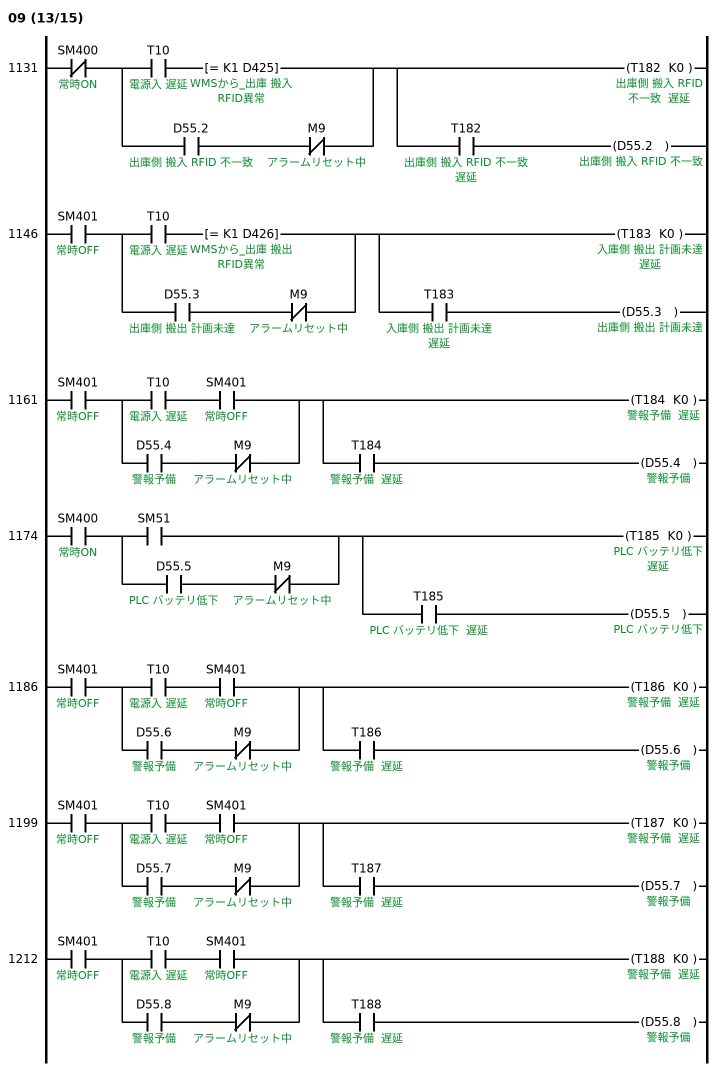
1131  LDI     SM400  ; 常時ON
      LD      T10  ; 電源入 遅延
      AND=    K1 D425  ; WMSから_出庫 搬入 RFID異常
      LD      D55.2  ; 出庫側 搬入 RFID 不一致
      ANI     M9  ; アラームリセット中
      ORB
      ANB
      OUT     T182 K0  ; 出庫側 搬入 RFID 不一致  遅延
      AND     T182  ; 出庫側 搬入 RFID 不一致  遅延
      OUT     D55.2  ; 出庫側 搬入 RFID 不一致
1146  LD      SM401  ; 常時OFF
      LD      T10  ; 電源入 遅延
      AND=    K1 D426  ; WMSから_出庫 搬出 RFID異常
      LD      D55.3  ; 出庫側 搬出 計画未達
      ANI     M9  ; アラームリセット中
      ORB
      ANB
      OUT     T183 K0  ; 入庫側 搬出 計画未達  遅延
      AND     T183  ; 入庫側 搬出 計画未達  遅延
      OUT     D55.3  ; 出庫側 搬出 計画未達
1161  LD      SM401  ; 常時OFF
      LD      T10  ; 電源入 遅延
      AND     SM401  ; 常時OFF
      LD      D55.4  ; 警報予備
      ANI     M9  ; アラームリセット中
      ORB
      ANB
      OUT     T184 K0  ; 警報予備  遅延
      AND     T184  ; 警報予備  遅延
      OUT     D55.4  ; 警報予備
1174  LD      SM400  ; 常時ON
      LD      SM51
      LD      D55.5  ; PLC バッテリ低下
      ANI     M9  ; アラームリセット中
      ORB
      ANB
      OUT     T185 K0  ; PLC バッテリ低下  遅延
      AND     T185  ; PLC バッテリ低下  遅延
      OUT     D55.5  ; PLC バッテリ低下
1186  LD      SM401  ; 常時OFF
      LD      T10  ; 電源入 遅延
      AND     SM401  ; 常時OFF
      LD      D55.6  ; 警報予備
      ANI     M9  ; アラームリセット中
      ORB
      ANB
      OUT     T186 K0  ; 警報予備  遅延
      AND     T186  ; 警報予備  遅延
      OUT     D55.6  ; 警報予備
1199  LD      SM401  ; 常時OFF
      LD      T10  ; 電源入 遅延
      AND     SM401  ; 常時OFF
      LD      D55.7  ; 警報予備
      ANI     M9  ; アラームリセット中
      ORB
      ANB
      OUT     T187 K0  ; 警報予備  遅延
      AND     T187  ; 警報予備  遅延
      OUT     D55.7  ; 警報予備
1212  LD      SM401  ; 常時OFF
      LD      T10  ; 電源入 遅延
      AND     SM401  ; 常時OFF
      LD      D55.8  ; 警報予備
      ANI     M9  ; アラームリセット中
      ORB
      ANB
      OUT     T188 K0  ; 警報予備  遅延
      AND     T188  ; 警報予備  遅延
      OUT     D55.8  ; 警報予備
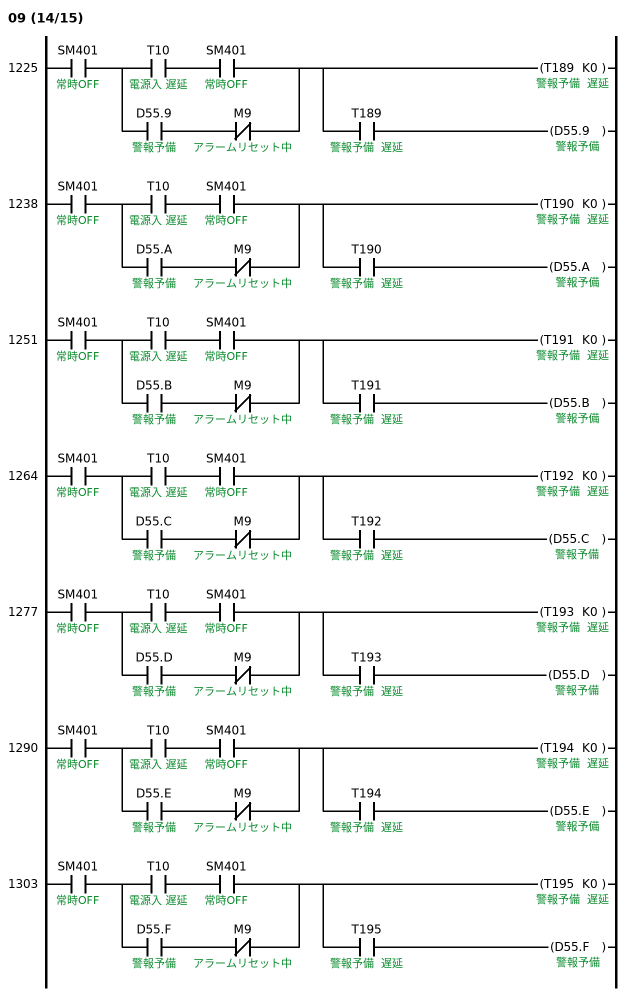
1225  LD      SM401  ; 常時OFF
      LD      T10  ; 電源入 遅延
      AND     SM401  ; 常時OFF
      LD      D55.9  ; 警報予備
      ANI     M9  ; アラームリセット中
      ORB
      ANB
      OUT     T189 K0  ; 警報予備  遅延
      AND     T189  ; 警報予備  遅延
      OUT     D55.9  ; 警報予備
1238  LD      SM401  ; 常時OFF
      LD      T10  ; 電源入 遅延
      AND     SM401  ; 常時OFF
      LD      D55.A  ; 警報予備
      ANI     M9  ; アラームリセット中
      ORB
      ANB
      OUT     T190 K0  ; 警報予備  遅延
      AND     T190  ; 警報予備  遅延
      OUT     D55.A  ; 警報予備
1251  LD      SM401  ; 常時OFF
      LD      T10  ; 電源入 遅延
      AND     SM401  ; 常時OFF
      LD      D55.B  ; 警報予備
      ANI     M9  ; アラームリセット中
      ORB
      ANB
      OUT     T191 K0  ; 警報予備  遅延
      AND     T191  ; 警報予備  遅延
      OUT     D55.B  ; 警報予備
1264  LD      SM401  ; 常時OFF
      LD      T10  ; 電源入 遅延
      AND     SM401  ; 常時OFF
      LD      D55.C  ; 警報予備
      ANI     M9  ; アラームリセット中
      ORB
      ANB
      OUT     T192 K0  ; 警報予備  遅延
      AND     T192  ; 警報予備  遅延
      OUT     D55.C  ; 警報予備
1277  LD      SM401  ; 常時OFF
      LD      T10  ; 電源入 遅延
      AND     SM401  ; 常時OFF
      LD      D55.D  ; 警報予備
      ANI     M9  ; アラームリセット中
      ORB
      ANB
      OUT     T193 K0  ; 警報予備  遅延
      AND     T193  ; 警報予備  遅延
      OUT     D55.D  ; 警報予備
1290  LD      SM401  ; 常時OFF
      LD      T10  ; 電源入 遅延
      AND     SM401  ; 常時OFF
      LD      D55.E  ; 警報予備
      ANI     M9  ; アラームリセット中
      ORB
      ANB
      OUT     T194 K0  ; 警報予備  遅延
      AND     T194  ; 警報予備  遅延
      OUT     D55.E  ; 警報予備
1303  LD      SM401  ; 常時OFF
      LD      T10  ; 電源入 遅延
      AND     SM401  ; 常時OFF
      LD      D55.F  ; 警報予備
      ANI     M9  ; アラームリセット中
      ORB
      ANB
      OUT     T195 K0  ; 警報予備  遅延
      AND     T195  ; 警報予備  遅延
      OUT     D55.F  ; 警報予備
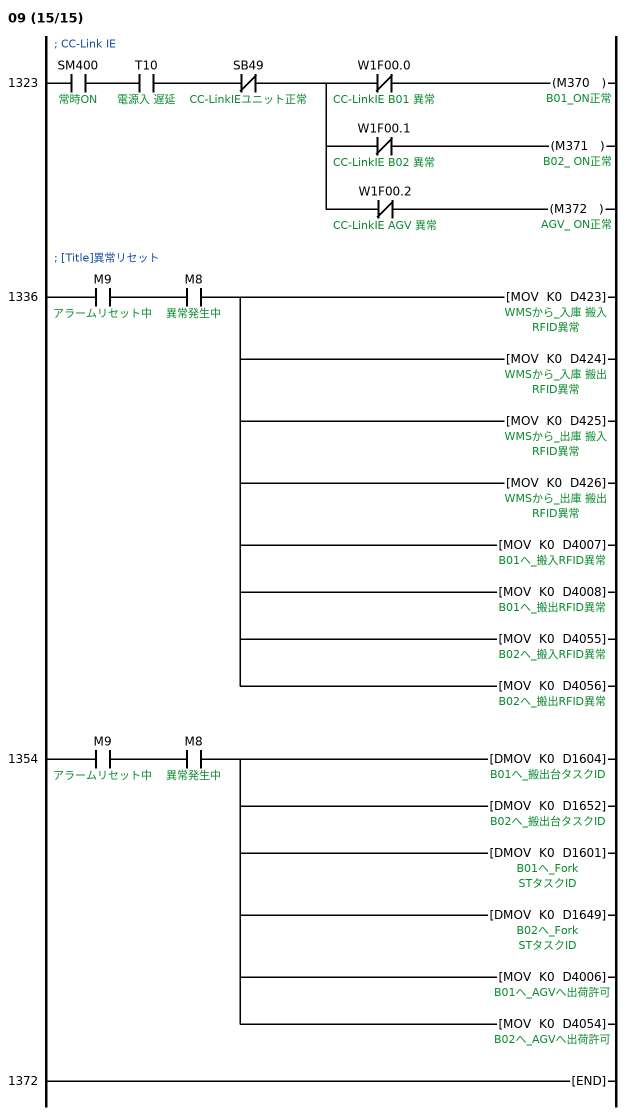
; CC-Link IE
1323  LD      SM400  ; 常時ON
      AND     T10  ; 電源入 遅延
      ANI     SB49  ; CC-LinkIEユニット正常
      MPS
      ANI     W1F00.0  ; CC-LinkIE B01 異常
      OUT     M370  ; B01_ON正常
      MRD
      ANI     W1F00.1  ; CC-LinkIE B02 異常
      OUT     M371  ; B02_ ON正常
      MPP
      ANI     W1F00.2  ; CC-LinkIE AGV 異常
      OUT     M372  ; AGV_ ON正常
; [Title]異常リセット
1336  LD      M9  ; アラームリセット中
      AND     M8  ; 異常発生中
      MOV     K0 D423
      MOV     K0 D424
      MOV     K0 D425
      MOV     K0 D426
      MOV     K0 D4007  ; B01へ_搬入RFID異常
      MOV     K0 D4008  ; B01へ_搬出RFID異常
      MOV     K0 D4055  ; B02へ_搬入RFID異常
      MOV     K0 D4056  ; B02へ_搬出RFID異常
1354  LD      M9  ; アラームリセット中
      AND     M8  ; 異常発生中
      DMOV    K0 D1604  ; B01へ_搬出台タスクID
      DMOV    K0 D1652  ; B02へ_搬出台タスクID
      DMOV    K0 D1601  ; B01へ_ForkSTタスクID
      DMOV    K0 D1649  ; B02へ_ForkSTタスクID
      MOV     K0 D4006  ; B01へ_AGVへ出荷許可
      MOV     K0 D4054  ; B02へ_AGVへ出荷許可
1372  END
END_PROGRAM

PROGRAM 10  // MAIN
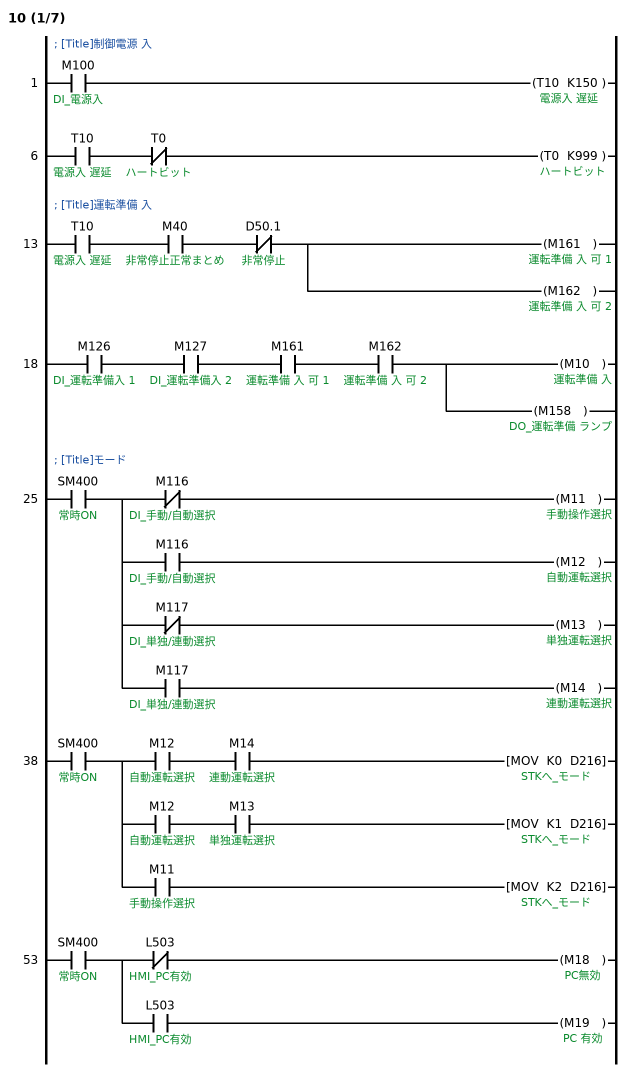
; [Title]制御電源 入
1     LD      M100  ; DI_電源入
      OUT     T10 K150  ; 電源入 遅延
6     LD      T10  ; 電源入 遅延
      ANI     T0  ; ハートビット
      OUT     T0 K999  ; ハートビット
; [Title]運転準備 入
13    LD      T10  ; 電源入 遅延
      AND     M40  ; 非常停止正常まとめ
      ANI     D50.1  ; 非常停止
      OUT     M161  ; 運転準備 入 可 1
      OUT     M162  ; 運転準備 入 可 2
18    LD      M126  ; DI_運転準備入 1
      AND     M127  ; DI_運転準備入 2
      AND     M161  ; 運転準備 入 可 1
      AND     M162  ; 運転準備 入 可 2
      OUT     M10  ; 運転準備 入
      OUT     M158  ; DO_運転準備 ランプ
; [Title]モード
25    LD      SM400  ; 常時ON
      MPS
      ANI     M116  ; DI_手動/自動選択
      OUT     M11  ; 手動操作選択
      MRD
      AND     M116  ; DI_手動/自動選択
      OUT     M12  ; 自動運転選択
      MRD
      ANI     M117  ; DI_単独/連動選択
      OUT     M13  ; 単独運転選択
      MPP
      AND     M117  ; DI_単独/連動選択
      OUT     M14  ; 連動運転選択
38    LD      SM400  ; 常時ON
      MPS
      AND     M12  ; 自動運転選択
      AND     M14  ; 連動運転選択
      MOV     K0 D216  ; STKへ_モード
      MRD
      AND     M12  ; 自動運転選択
      AND     M13  ; 単独運転選択
      MOV     K1 D216
      MPP
      AND     M11  ; 手動操作選択
      MOV     K2 D216
53    LD      SM400  ; 常時ON
      MPS
      ANI     L503  ; HMI_PC有効
      OUT     M18  ; PC無効
      MPP
      AND     L503  ; HMI_PC有効
      OUT     M19  ; PC 有効
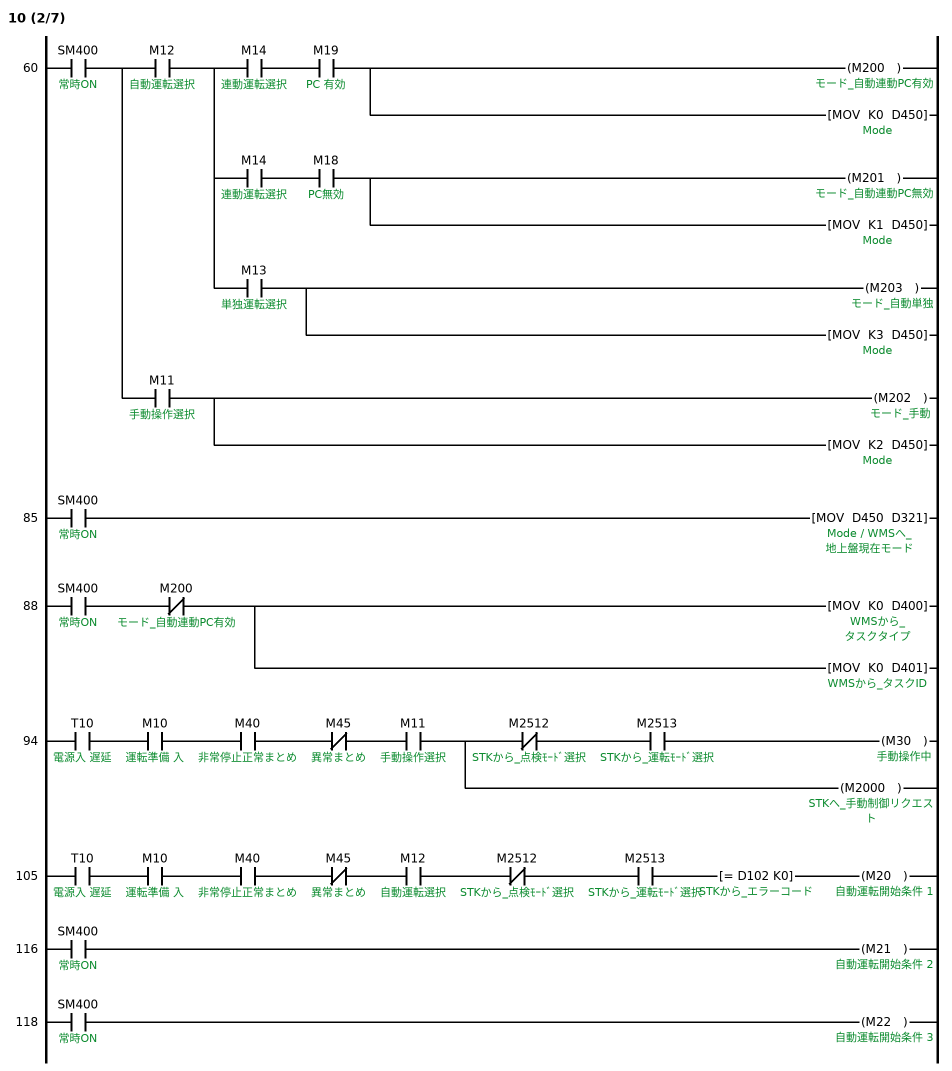
60    LD      SM400  ; 常時ON
      MPS
      AND     M12  ; 自動運転選択
      MPS
      AND     M14  ; 連動運転選択
      AND     M19  ; PC 有効
      OUT     M200  ; モード_自動連動PC有効
      MOV     K0 D450  ; Mode
      MRD
      AND     M14  ; 連動運転選択
      AND     M18  ; PC無効
      OUT     M201  ; モード_自動連動PC無効
      MOV     K1 D450
      MPP
      AND     M13  ; 単独運転選択
      OUT     M203  ; モード_自動単独
      MOV     K3 D450
      MPP
      AND     M11  ; 手動操作選択
      OUT     M202  ; モード_手動
      MOV     K2 D450
85    LD      SM400  ; 常時ON
      MOV     D450 D321  ; WMSへ_地上盤現在モード
88    LD      SM400  ; 常時ON
      ANI     M200  ; モード_自動連動PC有効
      MOV     K0 D400  ; WMSから_タスクタイプ
      MOV     K0 D401  ; WMSから_タスクID
94    LD      T10  ; 電源入 遅延
      AND     M10  ; 運転準備 入
      AND     M40  ; 非常停止正常まとめ
      ANI     M45  ; 異常まとめ
      AND     M11  ; 手動操作選択
      MPS
      ANI     M2512  ; STKから_点検ﾓｰﾄﾞ選択
      AND     M2513  ; STKから_運転ﾓｰﾄﾞ選択
      OUT     M30  ; 手動操作中
      MPP
      OUT     M2000  ; STKへ_手動制御リクエスト
105   LD      T10  ; 電源入 遅延
      AND     M10  ; 運転準備 入
      AND     M40  ; 非常停止正常まとめ
      ANI     M45  ; 異常まとめ
      AND     M12  ; 自動運転選択
      ANI     M2512  ; STKから_点検ﾓｰﾄﾞ選択
      AND     M2513  ; STKから_運転ﾓｰﾄﾞ選択
      AND=    D102 K0  ; STKから_エラーコード
      OUT     M20  ; 自動運転開始条件 1
116   LD      SM400  ; 常時ON
      OUT     M21  ; 自動運転開始条件 2
118   LD      SM400  ; 常時ON
      OUT     M22  ; 自動運転開始条件 3
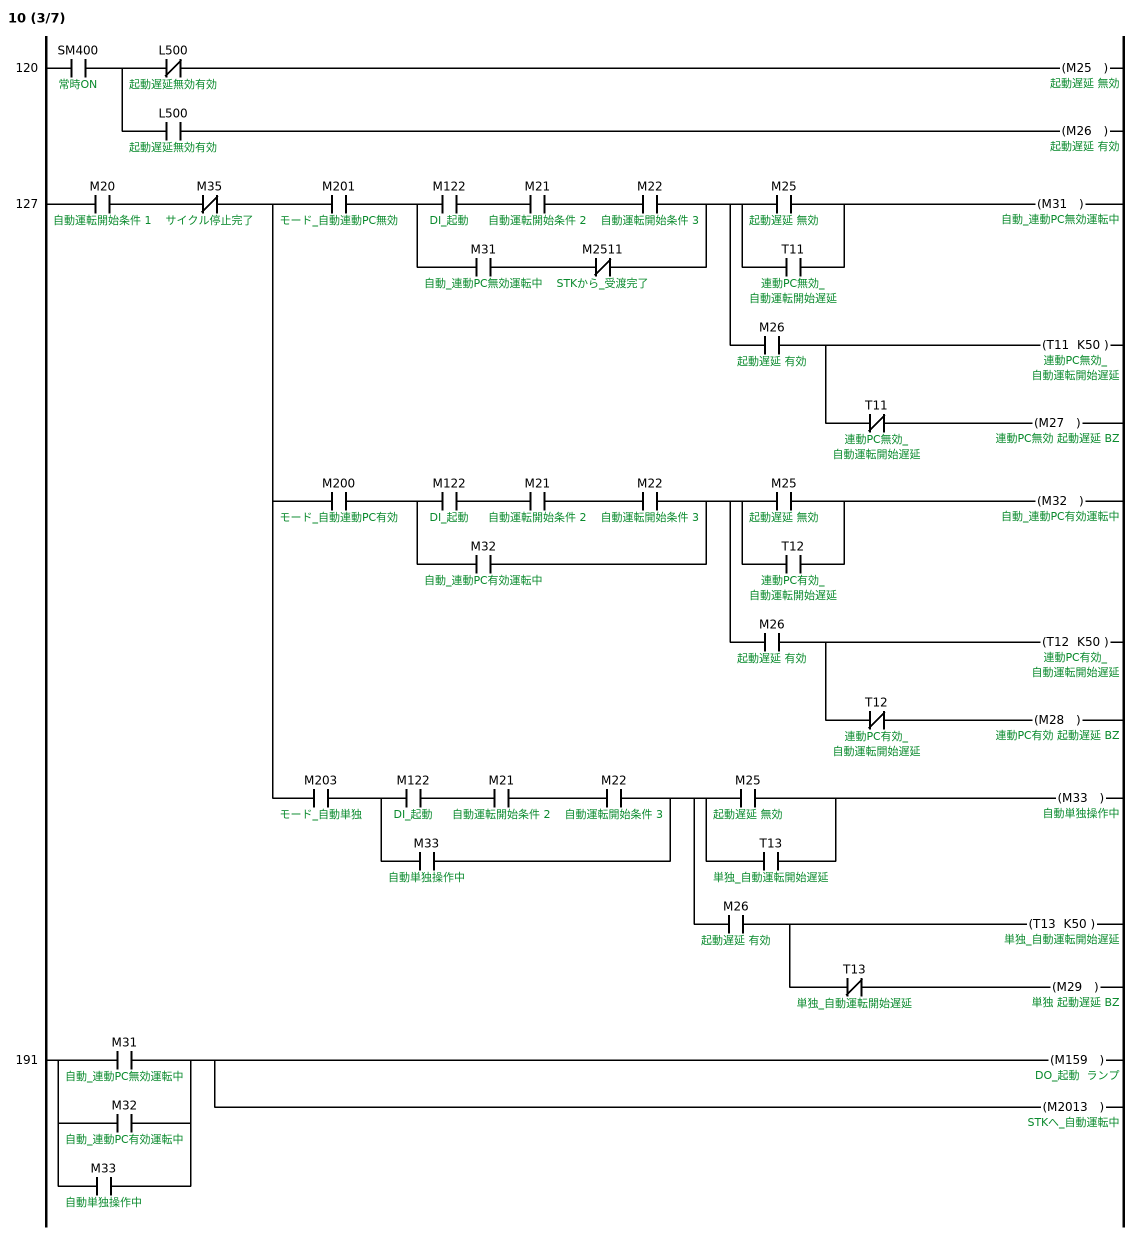
120   LD      SM400  ; 常時ON
      MPS
      ANI     L500  ; 起動遅延無効有効
      OUT     M25  ; 起動遅延 無効
      MPP
      AND     L500  ; 起動遅延無効有効
      OUT     M26  ; 起動遅延 有効
127   LD      M20  ; 自動運転開始条件 1
      ANI     M35  ; サイクル停止完了
      MPS
      AND     M201  ; モード_自動連動PC無効
      LD      M122  ; DI_起動
      AND     M21  ; 自動運転開始条件 2
      AND     M22  ; 自動運転開始条件 3
      LD      M31  ; 自動_連動PC無効運転中
      ANI     M2511  ; STKから_受渡完了
      ORB
      ANB
      MPS
      LD      M25  ; 起動遅延 無効
      OR      T11  ; 連動PC無効_自動運転開始遅延
      ANB
      OUT     M31  ; 自動_連動PC無効運転中
      MPP
      AND     M26  ; 起動遅延 有効
      OUT     T11 K50  ; 連動PC無効_自動運転開始遅延
      ANI     T11  ; 連動PC無効_自動運転開始遅延
      OUT     M27  ; 連動PC無効 起動遅延 BZ
      MRD
      AND     M200  ; モード_自動連動PC有効
      LD      M122  ; DI_起動
      AND     M21  ; 自動運転開始条件 2
      AND     M22  ; 自動運転開始条件 3
      OR      M32  ; 自動_連動PC有効運転中
      ANB
      MPS
      LD      M25  ; 起動遅延 無効
      OR      T12  ; 連動PC有効_自動運転開始遅延
      ANB
      OUT     M32  ; 自動_連動PC有効運転中
      MPP
      AND     M26  ; 起動遅延 有効
      OUT     T12 K50  ; 連動PC有効_自動運転開始遅延
      ANI     T12  ; 連動PC有効_自動運転開始遅延
      OUT     M28  ; 連動PC有効 起動遅延 BZ
      MPP
      AND     M203  ; モード_自動単独
      LD      M122  ; DI_起動
      AND     M21  ; 自動運転開始条件 2
      AND     M22  ; 自動運転開始条件 3
      OR      M33  ; 自動単独操作中
      ANB
      MPS
      LD      M25  ; 起動遅延 無効
      OR      T13  ; 単独_自動運転開始遅延
      ANB
      OUT     M33  ; 自動単独操作中
      MPP
      AND     M26  ; 起動遅延 有効
      OUT     T13 K50  ; 単独_自動運転開始遅延
      ANI     T13  ; 単独_自動運転開始遅延
      OUT     M29  ; 単独 起動遅延 BZ
191   LD      M31  ; 自動_連動PC無効運転中
      OR      M32  ; 自動_連動PC有効運転中
      OR      M33  ; 自動単独操作中
      OUT     M159  ; DO_起動  ランプ
      OUT     M2013  ; STKへ_自動運転中
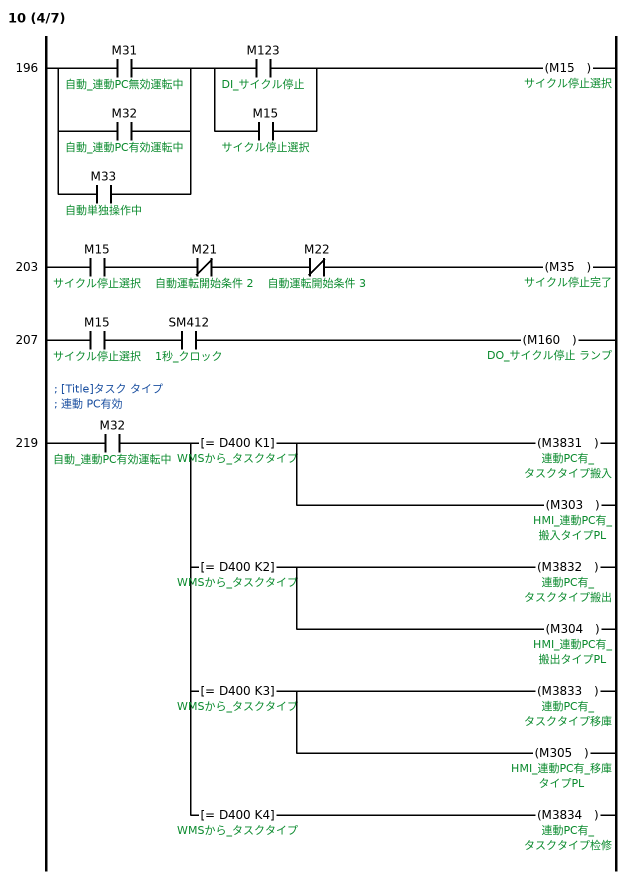
196   LD      M31  ; 自動_連動PC無効運転中
      OR      M32  ; 自動_連動PC有効運転中
      OR      M33  ; 自動単独操作中
      LD      M123  ; DI_サイクル停止
      OR      M15  ; サイクル停止選択
      ANB
      OUT     M15  ; サイクル停止選択
203   LD      M15  ; サイクル停止選択
      ANI     M21  ; 自動運転開始条件 2
      ANI     M22  ; 自動運転開始条件 3
      OUT     M35  ; サイクル停止完了
207   LD      M15  ; サイクル停止選択
      AND     SM412  ; 1秒_クロック
      OUT     M160  ; DO_サイクル停止 ランプ
; [Title]タスク タイプ
; 連動 PC有効
219   LD      M32  ; 自動_連動PC有効運転中
      MPS
      AND=    D400 K1  ; WMSから_タスクタイプ
      OUT     M3831  ; 連動PC有_タスクタイプ搬入
      OUT     M303  ; HMI_連動PC有_搬入タイプPL
      MRD
      AND=    D400 K2  ; WMSから_タスクタイプ
      OUT     M3832  ; 連動PC有_タスクタイプ搬出
      OUT     M304  ; HMI_連動PC有_搬出タイプPL
      MRD
      AND=    D400 K3  ; WMSから_タスクタイプ
      OUT     M3833  ; 連動PC有_タスクタイプ移庫
      OUT     M305  ; HMI_連動PC有_移庫 タイプPL
      MPP
      AND=    D400 K4  ; WMSから_タスクタイプ
      OUT     M3834  ; 連動PC有_タスクタイプ检修
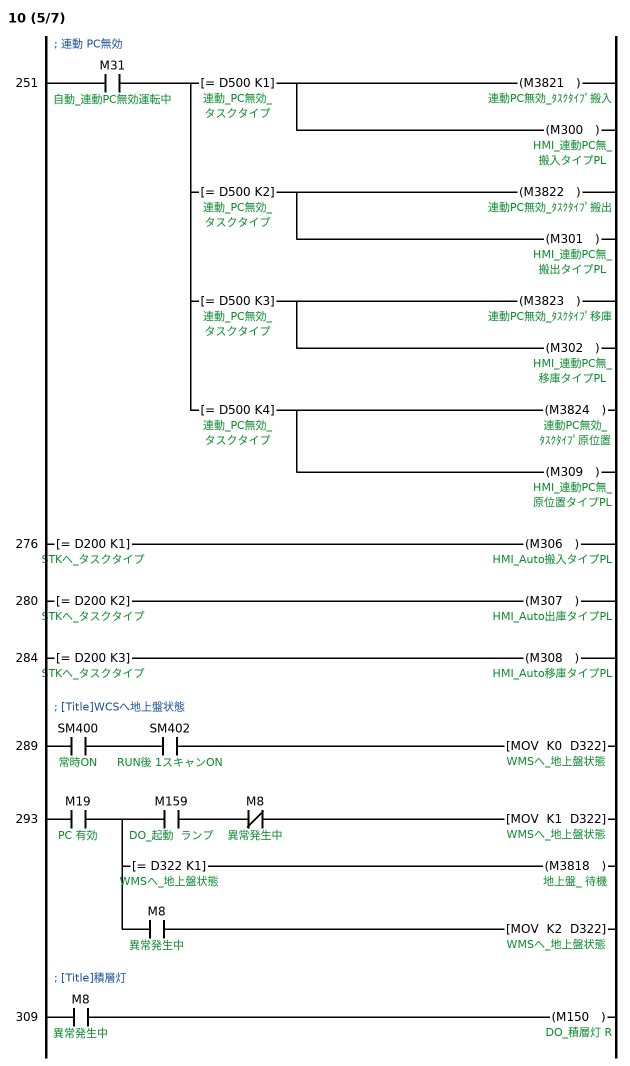
; 連動 PC無効
251   LD      M31  ; 自動_連動PC無効運転中
      MPS
      AND=    D500 K1  ; 連動_PC無効_タスクタイプ
      OUT     M3821  ; 連動PC無効_ﾀｽｸﾀｲﾌﾟ搬入
      OUT     M300  ; HMI_連動PC無_搬入タイプPL
      MRD
      AND=    D500 K2  ; 連動_PC無効_タスクタイプ
      OUT     M3822  ; 連動PC無効_ﾀｽｸﾀｲﾌﾟ搬出
      OUT     M301  ; HMI_連動PC無_搬出タイプPL
      MRD
      AND=    D500 K3  ; 連動_PC無効_タスクタイプ
      OUT     M3823  ; 連動PC無効_ﾀｽｸﾀｲﾌﾟ移庫
      OUT     M302  ; HMI_連動PC無_移庫タイプPL
      MPP
      AND=    D500 K4  ; 連動_PC無効_タスクタイプ
      OUT     M3824  ; 連動PC無効_ﾀｽｸﾀｲﾌﾟ原位置
      OUT     M309  ; HMI_連動PC無_原位置タイプPL
276   LD=     D200 K1  ; STKへ_タスクタイプ
      OUT     M306  ; HMI_Auto搬入タイプPL
280   LD=     D200 K2  ; STKへ_タスクタイプ
      OUT     M307  ; HMI_Auto出庫タイプPL
284   LD=     D200 K3  ; STKへ_タスクタイプ
      OUT     M308  ; HMI_Auto移庫タイプPL
; [Title]WCSへ地上盤状態
289   LD      SM400  ; 常時ON
      AND     SM402  ; RUN後 1スキャンON
      MOV     K0 D322  ; WMSへ_地上盤状態
293   LD      M19  ; PC 有効
      MPS
      AND     M159  ; DO_起動  ランプ
      ANI     M8  ; 異常発生中
      MOV     K1 D322
      MRD
      AND=    D322 K1  ; WMSへ_地上盤状態
      OUT     M3818  ; 地上盤_ 待機
      MPP
      AND     M8  ; 異常発生中
      MOV     K2 D322
; [Title]積層灯
309   LD      M8  ; 異常発生中
      OUT     M150  ; DO_積層灯 R
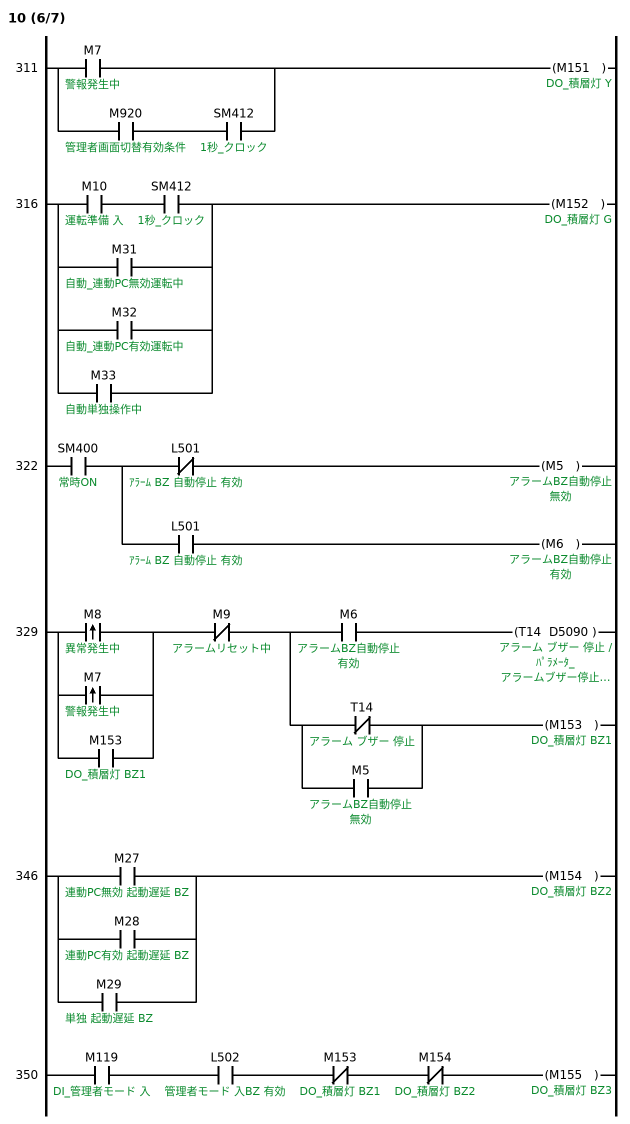
311   LD      M7  ; 警報発生中
      LD      M920  ; 管理者画面切替有効条件
      AND     SM412  ; 1秒_クロック
      ORB
      OUT     M151  ; DO_積層灯 Y
316   LD      M10  ; 運転準備 入
      AND     SM412  ; 1秒_クロック
      OR      M31  ; 自動_連動PC無効運転中
      OR      M32  ; 自動_連動PC有効運転中
      OR      M33  ; 自動単独操作中
      OUT     M152  ; DO_積層灯 G
322   LD      SM400  ; 常時ON
      MPS
      ANI     L501  ; ｱﾗｰﾑ BZ 自動停止 有効
      OUT     M5  ; アラームBZ自動停止 無効
      MPP
      AND     L501  ; ｱﾗｰﾑ BZ 自動停止 有効
      OUT     M6  ; アラームBZ自動停止 有効
329   LDP     M8  ; 異常発生中
      ORP     M7  ; 警報発生中
      OR      M153  ; DO_積層灯 BZ1
      ANI     M9  ; アラームリセット中
      MPS
      AND     M6  ; アラームBZ自動停止 有効
      OUT     T14 D5090  ; アラーム ブザー 停止 / ﾊﾟﾗﾒｰﾀ_アラームブザー停止設定値
      MPP
      LDI     T14  ; アラーム ブザー 停止
      OR      M5  ; アラームBZ自動停止 無効
      ANB
      OUT     M153  ; DO_積層灯 BZ1
346   LD      M27  ; 連動PC無効 起動遅延 BZ
      OR      M28  ; 連動PC有効 起動遅延 BZ
      OR      M29  ; 単独 起動遅延 BZ
      OUT     M154  ; DO_積層灯 BZ2
350   LD      M119  ; DI_管理者モード 入
      AND     L502  ; 管理者モード 入BZ 有効
      ANI     M153  ; DO_積層灯 BZ1
      ANI     M154  ; DO_積層灯 BZ2
      OUT     M155  ; DO_積層灯 BZ3
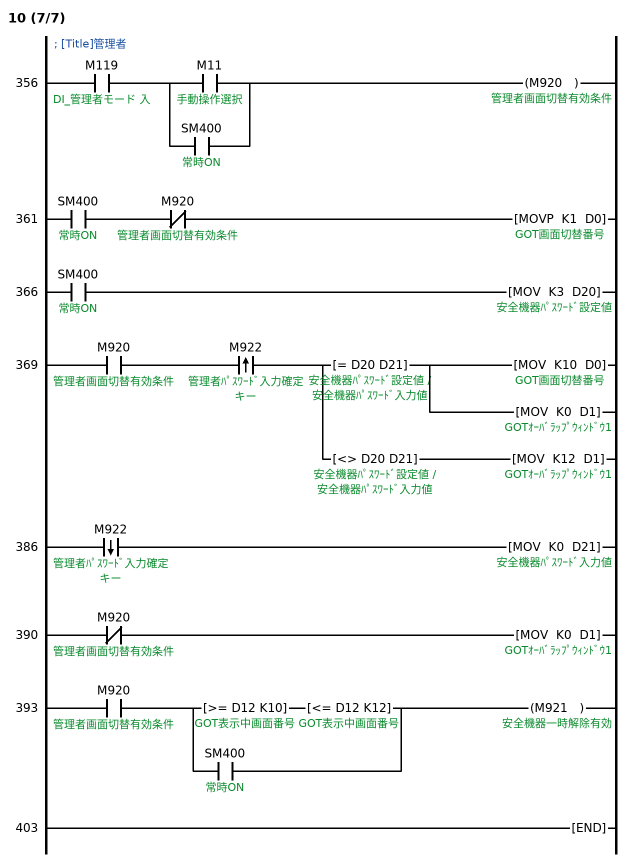
; [Title]管理者
356   LD      M119  ; DI_管理者モード 入
      LD      M11  ; 手動操作選択
      OR      SM400  ; 常時ON
      ANB
      OUT     M920  ; 管理者画面切替有効条件
361   LD      SM400  ; 常時ON
      ANI     M920  ; 管理者画面切替有効条件
      MOVP    K1 D0  ; GOT画面切替番号
366   LD      SM400  ; 常時ON
      MOV     K3 D20  ; 安全機器ﾊﾟｽﾜｰﾄﾞ設定値
369   LD      M920  ; 管理者画面切替有効条件
      ANDP    M922  ; 管理者ﾊﾟｽﾜｰﾄﾞ入力確定キー
      MPS
      AND=    D20 D21  ; 安全機器ﾊﾟｽﾜｰﾄﾞ設定値 / 安全機器ﾊﾟｽﾜｰﾄﾞ入力値
      MOV     K10 D0
      MOV     K0 D1  ; GOTｵｰﾊﾞﾗｯﾌﾟｳｨﾝﾄﾞｳ1
      MPP
      AND<>   D20 D21  ; 安全機器ﾊﾟｽﾜｰﾄﾞ設定値 / 安全機器ﾊﾟｽﾜｰﾄﾞ入力値
      MOV     K12 D1
386   LDF     M922  ; 管理者ﾊﾟｽﾜｰﾄﾞ入力確定キー
      MOV     K0 D21
390   LDI     M920  ; 管理者画面切替有効条件
      MOV     K0 D1
393   LD      M920  ; 管理者画面切替有効条件
      LD>=    D12 K10  ; GOT表示中画面番号
      AND<=   D12 K12  ; GOT表示中画面番号
      OR      SM400  ; 常時ON
      ANB
      OUT     M921  ; 安全機器一時解除有効
403   END
END_PROGRAM

PROGRAM 11  // STK 自動/連動 PC有効モード
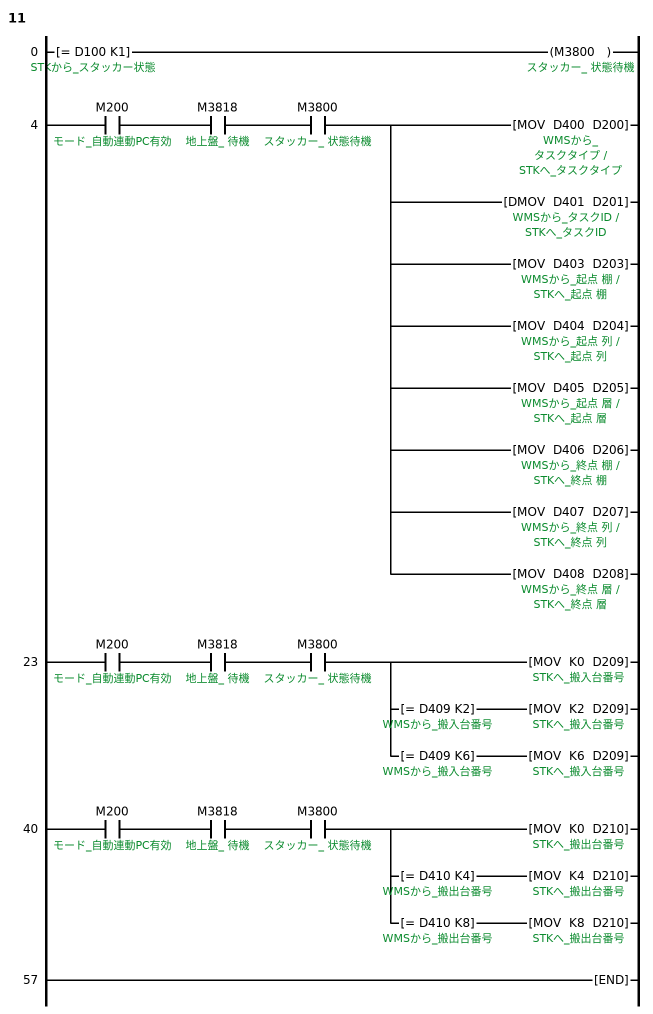
0     LD=     D100 K1  ; STKから_スタッカー状態
      OUT     M3800  ; スタッカー_ 状態待機
4     LD      M200  ; モード_自動連動PC有効
      AND     M3818  ; 地上盤_ 待機
      AND     M3800  ; スタッカー_ 状態待機
      MOV     D400 D200  ; WMSから_タスクタイプ / STKへ_タスクタイプ
      DMOV    D401 D201  ; WMSから_タスクID / STKへ_タスクID
      MOV     D403 D203  ; WMSから_起点 棚 / STKへ_起点 棚
      MOV     D404 D204  ; WMSから_起点 列 / STKへ_起点 列
      MOV     D405 D205  ; WMSから_起点 層 / STKへ_起点 層
      MOV     D406 D206  ; WMSから_終点 棚 / STKへ_終点 棚
      MOV     D407 D207  ; WMSから_終点 列 / STKへ_終点 列
      MOV     D408 D208  ; WMSから_終点 層 / STKへ_終点 層
23    LD      M200  ; モード_自動連動PC有効
      AND     M3818  ; 地上盤_ 待機
      AND     M3800  ; スタッカー_ 状態待機
      MOV     K0 D209  ; STKへ_搬入台番号
      MPS
      AND=    D409 K2  ; WMSから_搬入台番号
      MOV     K2 D209
      MPP
      AND=    D409 K6  ; WMSから_搬入台番号
      MOV     K6 D209
40    LD      M200  ; モード_自動連動PC有効
      AND     M3818  ; 地上盤_ 待機
      AND     M3800  ; スタッカー_ 状態待機
      MOV     K0 D210  ; STKへ_搬出台番号
      MPS
      AND=    D410 K4  ; WMSから_搬出台番号
      MOV     K4 D210
      MPP
      AND=    D410 K8  ; WMSから_搬出台番号
      MOV     K8 D210
57    END
END_PROGRAM

PROGRAM 12  // STK 自動/連動PC 無効モード
VAR
  __IST_02f34114d45741f9 : I+ST_02f34114d45741f9;
  __IST_08ba2391820a4452 : I+ST_08ba2391820a4452;
END_VAR
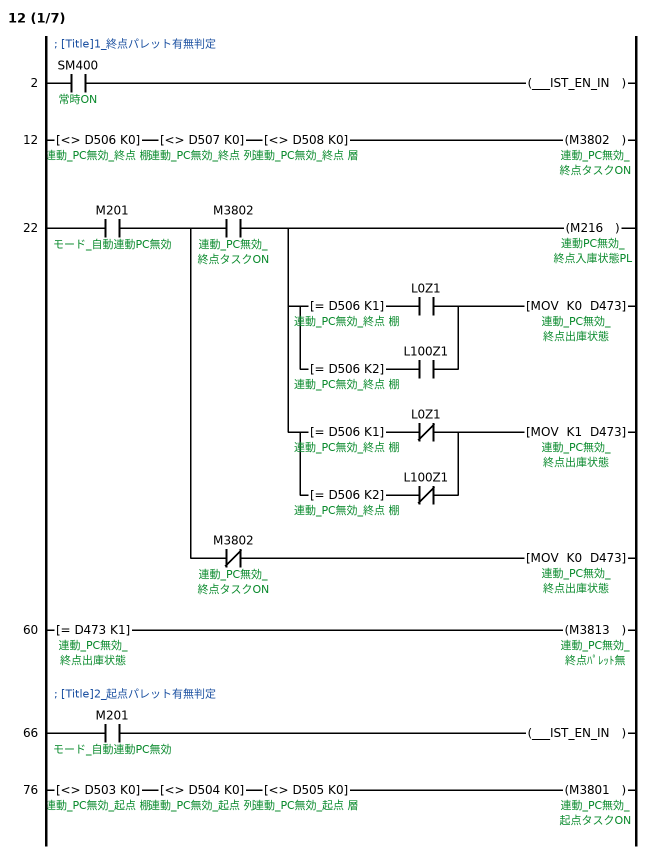
; FB BLK START I+ST_08ba2391820a4452(__IST_08ba2391820a4452)
; [Title]1_終点パレット有無判定
2     LD      SM400  ; 常時ON
      OUT     ___IST_EN_IN
; FB START
; FB_NAME I+ST_08ba2391820a4452
; INSTANCE_NAME __IST_08ba2391820a4452
; FB IN_B:__IST_EN_IN
; FB OUT___IST_EN_OUT:B
; FB END
; FB BLK END
12    LD<>    D506 K0  ; 連動_PC無効_終点 棚
      AND<>   D507 K0  ; 連動_PC無効_終点 列
      AND<>   D508 K0  ; 連動_PC無効_終点 層
      OUT     M3802  ; 連動_PC無効_終点タスクON
22    LD      M201  ; モード_自動連動PC無効
      MPS
      AND     M3802  ; 連動_PC無効_終点タスクON
      OUT     M216  ; 連動PC無効_終点入庫状態PL
      MPS
      LD=     D506 K1  ; 連動_PC無効_終点 棚
      AND     L0Z1
      LD=     D506 K2  ; 連動_PC無効_終点 棚
      AND     L100Z1
      ORB
      ANB
      MOV     K0 D473  ; 連動_PC無効_終点出庫状態
      MPP
      LD=     D506 K1  ; 連動_PC無効_終点 棚
      ANI     L0Z1
      LD=     D506 K2  ; 連動_PC無効_終点 棚
      ANI     L100Z1
      ORB
      ANB
      MOV     K1 D473
      MPP
      ANI     M3802  ; 連動_PC無効_終点タスクON
      MOV     K0 D473
60    LD=     D473 K1  ; 連動_PC無効_終点出庫状態
      OUT     M3813  ; 連動_PC無効_終点ﾊﾟﾚｯﾄ無
; FB BLK START I+ST_02f34114d45741f9(__IST_02f34114d45741f9)
; [Title]2_起点パレット有無判定
66    LD      M201  ; モード_自動連動PC無効
      OUT     ___IST_EN_IN
; FB START
; FB_NAME I+ST_02f34114d45741f9
; INSTANCE_NAME __IST_02f34114d45741f9
; FB IN_B:__IST_EN_IN
; FB OUT___IST_EN_OUT:B
; FB END
; FB BLK END
76    LD<>    D503 K0  ; 連動_PC無効_起点 棚
      AND<>   D504 K0  ; 連動_PC無効_起点 列
      AND<>   D505 K0  ; 連動_PC無効_起点 層
      OUT     M3801  ; 連動_PC無効_起点タスクON
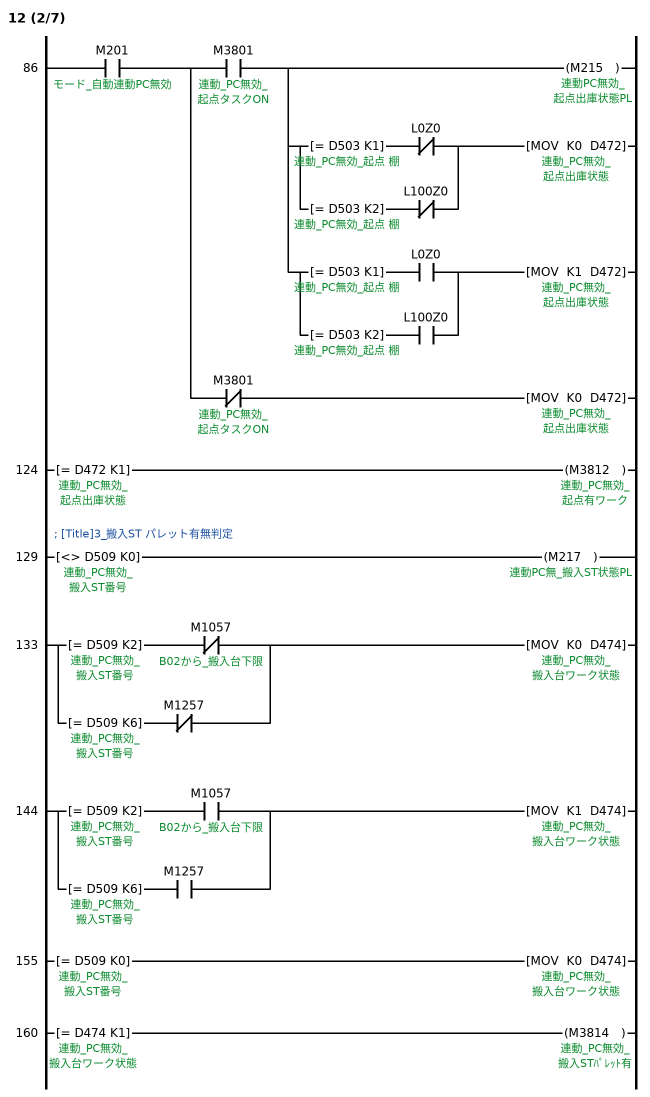
86    LD      M201  ; モード_自動連動PC無効
      MPS
      AND     M3801  ; 連動_PC無効_起点タスクON
      OUT     M215  ; 連動PC無効_起点出庫状態PL
      MPS
      LD=     D503 K1  ; 連動_PC無効_起点 棚
      ANI     L0Z0
      LD=     D503 K2  ; 連動_PC無効_起点 棚
      ANI     L100Z0
      ORB
      ANB
      MOV     K0 D472  ; 連動_PC無効_起点出庫状態
      MPP
      LD=     D503 K1  ; 連動_PC無効_起点 棚
      AND     L0Z0
      LD=     D503 K2  ; 連動_PC無効_起点 棚
      AND     L100Z0
      ORB
      ANB
      MOV     K1 D472
      MPP
      ANI     M3801  ; 連動_PC無効_起点タスクON
      MOV     K0 D472
124   LD=     D472 K1  ; 連動_PC無効_起点出庫状態
      OUT     M3812  ; 連動_PC無効_起点有ワーク
; [Title]3_搬入ST パレット有無判定
129   LD<>    D509 K0  ; 連動_PC無効_搬入ST番号
      OUT     M217  ; 連動PC無_搬入ST状態PL
133   LD=     D509 K2  ; 連動_PC無効_搬入ST番号
      ANI     M1057  ; B02から_搬入台下限
      LD=     D509 K6  ; 連動_PC無効_搬入ST番号
      ANI     M1257
      ORB
      MOV     K0 D474  ; 連動_PC無効_搬入台ワーク状態
144   LD=     D509 K2  ; 連動_PC無効_搬入ST番号
      AND     M1057  ; B02から_搬入台下限
      LD=     D509 K6  ; 連動_PC無効_搬入ST番号
      AND     M1257
      ORB
      MOV     K1 D474
155   LD=     D509 K0  ; 連動_PC無効_搬入ST番号
      MOV     K0 D474
160   LD=     D474 K1  ; 連動_PC無効_搬入台ワーク状態
      OUT     M3814  ; 連動_PC無効_搬入STﾊﾟﾚｯﾄ有
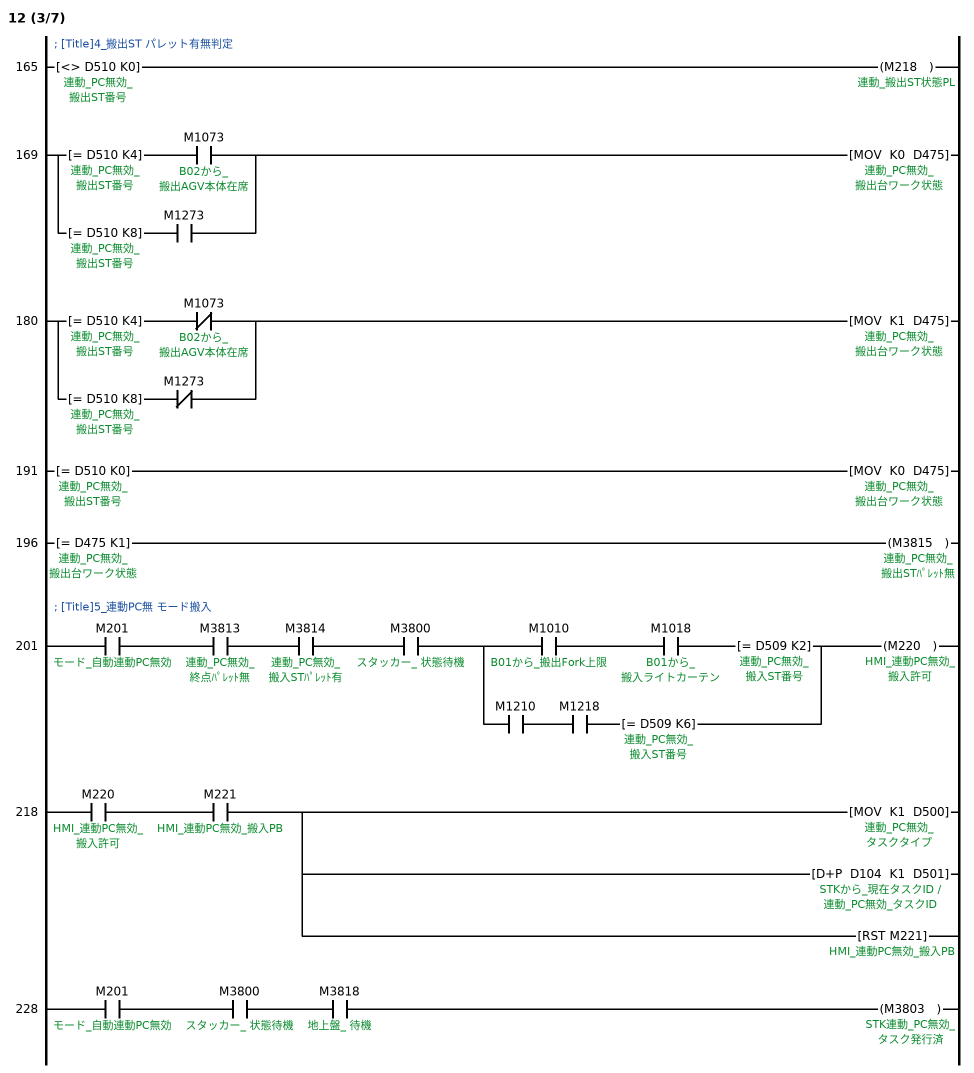
; [Title]4_搬出ST パレット有無判定
165   LD<>    D510 K0  ; 連動_PC無効_搬出ST番号
      OUT     M218  ; 連動_搬出ST状態PL
169   LD=     D510 K4  ; 連動_PC無効_搬出ST番号
      AND     M1073  ; B02から_搬出AGV本体在席
      LD=     D510 K8  ; 連動_PC無効_搬出ST番号
      AND     M1273
      ORB
      MOV     K0 D475  ; 連動_PC無効_搬出台ワーク状態
180   LD=     D510 K4  ; 連動_PC無効_搬出ST番号
      ANI     M1073  ; B02から_搬出AGV本体在席
      LD=     D510 K8  ; 連動_PC無効_搬出ST番号
      ANI     M1273
      ORB
      MOV     K1 D475
191   LD=     D510 K0  ; 連動_PC無効_搬出ST番号
      MOV     K0 D475
196   LD=     D475 K1  ; 連動_PC無効_搬出台ワーク状態
      OUT     M3815  ; 連動_PC無効_搬出STﾊﾟﾚｯﾄ無
; [Title]5_連動PC無 モード搬入
201   LD      M201  ; モード_自動連動PC無効
      AND     M3813  ; 連動_PC無効_終点ﾊﾟﾚｯﾄ無
      AND     M3814  ; 連動_PC無効_搬入STﾊﾟﾚｯﾄ有
      AND     M3800  ; スタッカー_ 状態待機
      LD      M1010  ; B01から_搬出Fork上限
      AND     M1018  ; B01から_搬入ライトカーテン
      AND=    D509 K2  ; 連動_PC無効_搬入ST番号
      LD      M1210
      AND     M1218
      AND=    D509 K6  ; 連動_PC無効_搬入ST番号
      ORB
      ANB
      OUT     M220  ; HMI_連動PC無効_搬入許可
218   LD      M220  ; HMI_連動PC無効_搬入許可
      AND     M221  ; HMI_連動PC無効_搬入PB
      MOV     K1 D500  ; 連動_PC無効_タスクタイプ
      D+P     D104 K1 D501  ; STKから_現在タスクID / 連動_PC無効_タスクID
      RST     M221  ; HMI_連動PC無効_搬入PB
228   LD      M201  ; モード_自動連動PC無効
      AND     M3800  ; スタッカー_ 状態待機
      AND     M3818  ; 地上盤_ 待機
      OUT     M3803  ; STK連動_PC無効_タスク発行済
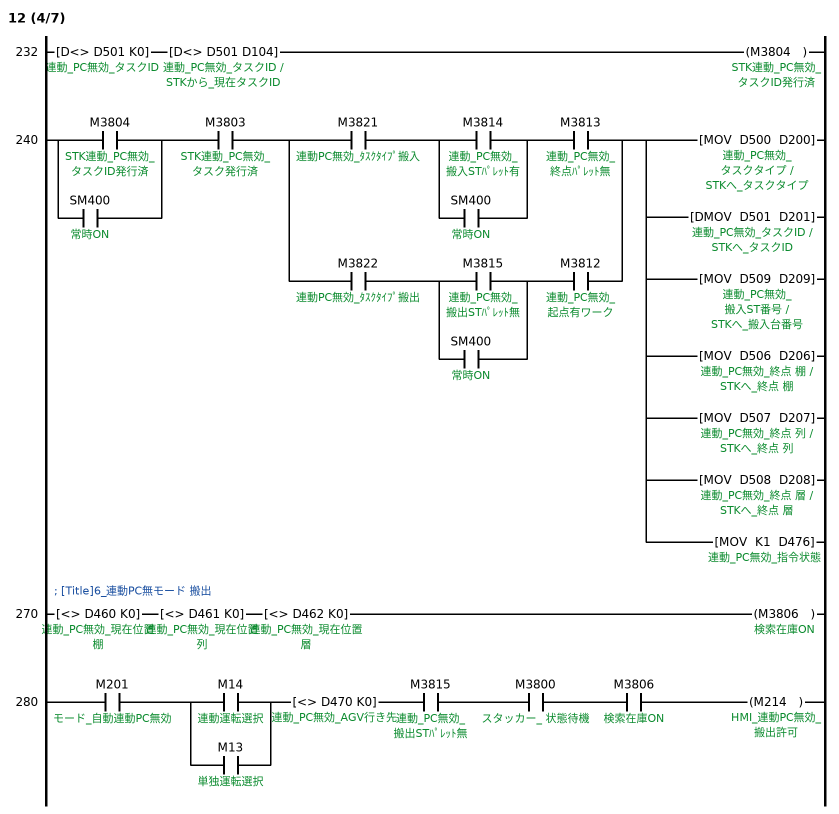
232   LDD<>   D501 K0  ; 連動_PC無効_タスクID
      ANDD<>  D501 D104  ; 連動_PC無効_タスクID / STKから_現在タスクID
      OUT     M3804  ; STK連動_PC無効_タスクID発行済
240   LD      M3804  ; STK連動_PC無効_タスクID発行済
      OR      SM400  ; 常時ON
      AND     M3803  ; STK連動_PC無効_タスク発行済
      LD      M3821  ; 連動PC無効_ﾀｽｸﾀｲﾌﾟ搬入
      LD      M3814  ; 連動_PC無効_搬入STﾊﾟﾚｯﾄ有
      OR      SM400  ; 常時ON
      ANB
      AND     M3813  ; 連動_PC無効_終点ﾊﾟﾚｯﾄ無
      LD      M3822  ; 連動PC無効_ﾀｽｸﾀｲﾌﾟ搬出
      LD      M3815  ; 連動_PC無効_搬出STﾊﾟﾚｯﾄ無
      OR      SM400  ; 常時ON
      ANB
      AND     M3812  ; 連動_PC無効_起点有ワーク
      ORB
      ANB
      MOV     D500 D200  ; STKへ_タスクタイプ
      DMOV    D501 D201  ; STKへ_タスクID
      MOV     D509 D209  ; STKへ_搬入台番号
      MOV     D506 D206  ; STKへ_終点 棚
      MOV     D507 D207  ; STKへ_終点 列
      MOV     D508 D208  ; STKへ_終点 層
      MOV     K1 D476  ; 連動_PC無効_指令状態
; [Title]6_連動PC無モード 搬出
270   LD<>    D460 K0  ; 連動_PC無効_現在位置 棚
      AND<>   D461 K0  ; 連動_PC無効_現在位置 列
      AND<>   D462 K0  ; 連動_PC無効_現在位置 層
      OUT     M3806  ; 検索在庫ON
280   LD      M201  ; モード_自動連動PC無効
      LD      M14  ; 連動運転選択
      OR      M13  ; 単独運転選択
      ANB
      AND<>   D470 K0  ; 連動_PC無効_AGV行き先
      AND     M3815  ; 連動_PC無効_搬出STﾊﾟﾚｯﾄ無
      AND     M3800  ; スタッカー_ 状態待機
      AND     M3806  ; 検索在庫ON
      OUT     M214  ; HMI_連動PC無効_搬出許可
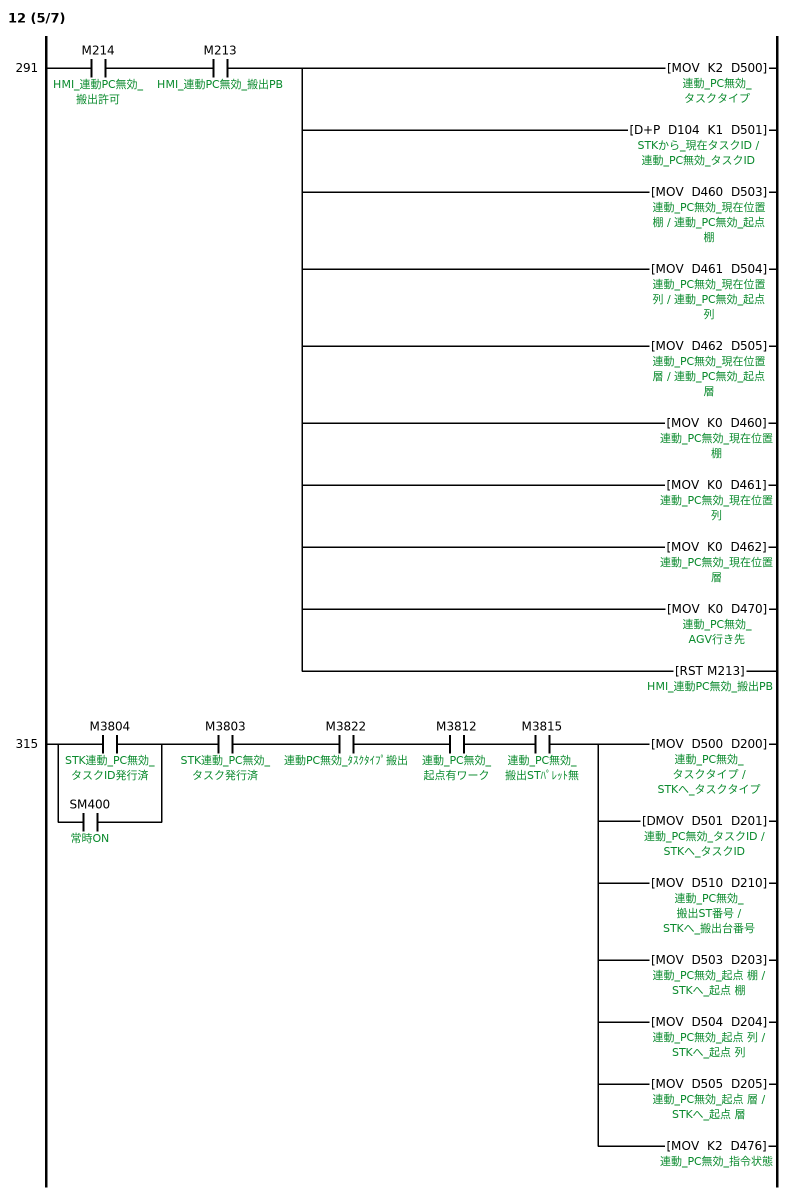
291   LD      M214  ; HMI_連動PC無効_搬出許可
      AND     M213  ; HMI_連動PC無効_搬出PB
      MOV     K2 D500
      D+P     D104 K1 D501
      MOV     D460 D503
      MOV     D461 D504
      MOV     D462 D505
      MOV     K0 D460
      MOV     K0 D461
      MOV     K0 D462
      MOV     K0 D470
      RST     M213  ; HMI_連動PC無効_搬出PB
315   LD      M3804  ; STK連動_PC無効_タスクID発行済
      OR      SM400  ; 常時ON
      AND     M3803  ; STK連動_PC無効_タスク発行済
      AND     M3822  ; 連動PC無効_ﾀｽｸﾀｲﾌﾟ搬出
      AND     M3812  ; 連動_PC無効_起点有ワーク
      AND     M3815  ; 連動_PC無効_搬出STﾊﾟﾚｯﾄ無
      MOV     D500 D200
      DMOV    D501 D201
      MOV     D510 D210  ; STKへ_搬出台番号
      MOV     D503 D203  ; STKへ_起点 棚
      MOV     D504 D204  ; STKへ_起点 列
      MOV     D505 D205  ; STKへ_起点 層
      MOV     K2 D476
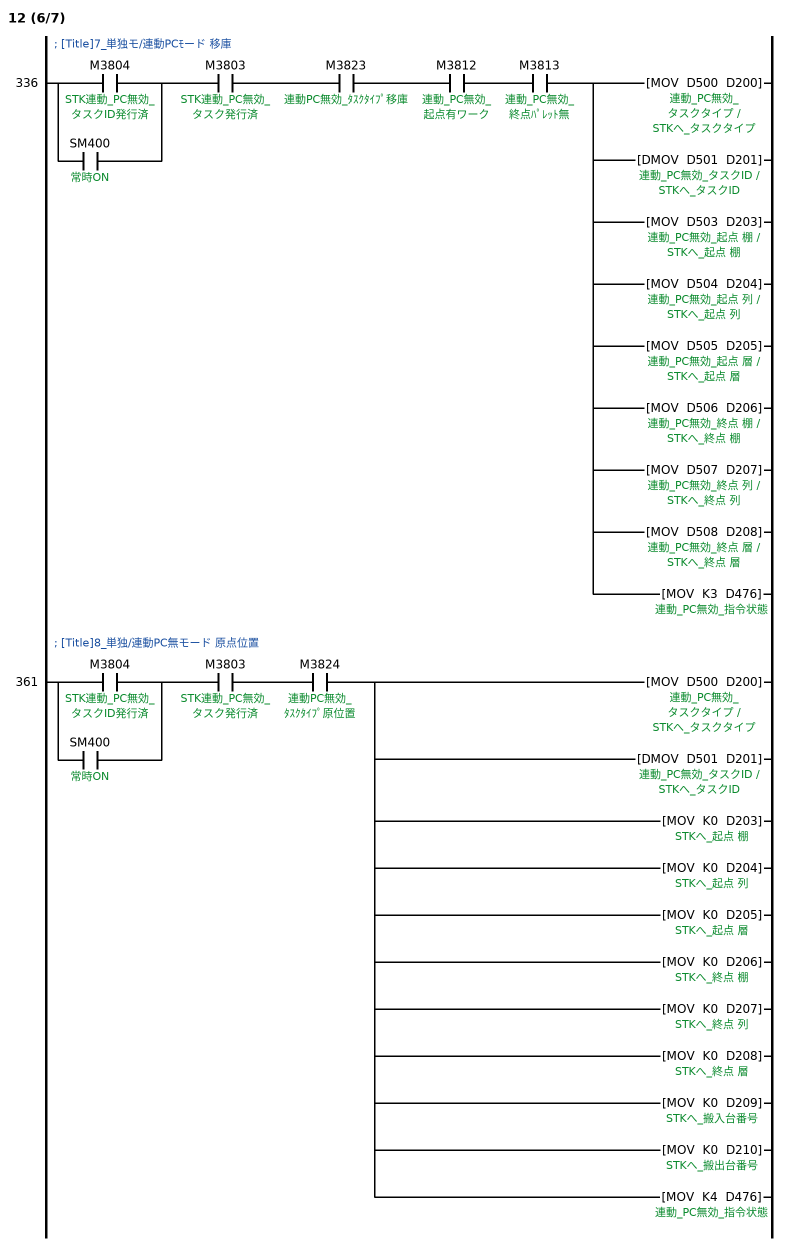
; [Title]7_単独モ/連動PCﾓード 移庫
336   LD      M3804  ; STK連動_PC無効_タスクID発行済
      OR      SM400  ; 常時ON
      AND     M3803  ; STK連動_PC無効_タスク発行済
      AND     M3823  ; 連動PC無効_ﾀｽｸﾀｲﾌﾟ移庫
      AND     M3812  ; 連動_PC無効_起点有ワーク
      AND     M3813  ; 連動_PC無効_終点ﾊﾟﾚｯﾄ無
      MOV     D500 D200
      DMOV    D501 D201
      MOV     D503 D203
      MOV     D504 D204
      MOV     D505 D205
      MOV     D506 D206
      MOV     D507 D207
      MOV     D508 D208
      MOV     K3 D476
; [Title]8_単独/連動PC無モード 原点位置
361   LD      M3804  ; STK連動_PC無効_タスクID発行済
      OR      SM400  ; 常時ON
      AND     M3803  ; STK連動_PC無効_タスク発行済
      AND     M3824  ; 連動PC無効_ﾀｽｸﾀｲﾌﾟ原位置
      MOV     D500 D200
      DMOV    D501 D201
      MOV     K0 D203
      MOV     K0 D204
      MOV     K0 D205
      MOV     K0 D206
      MOV     K0 D207
      MOV     K0 D208
      MOV     K0 D209
      MOV     K0 D210
      MOV     K4 D476
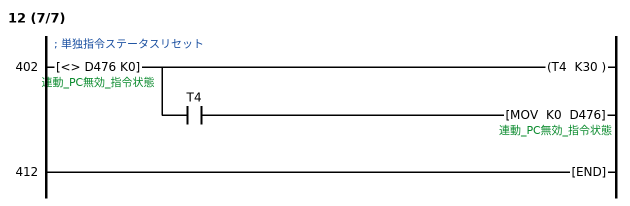
; 単独指令ステータスリセット
402   LD<>    D476 K0  ; 連動_PC無効_指令状態
      OUT     T4 K30
      AND     T4
      MOV     K0 D476
412   END
END_PROGRAM

PROGRAM 14  // STK 手動ﾓｰﾄﾞ
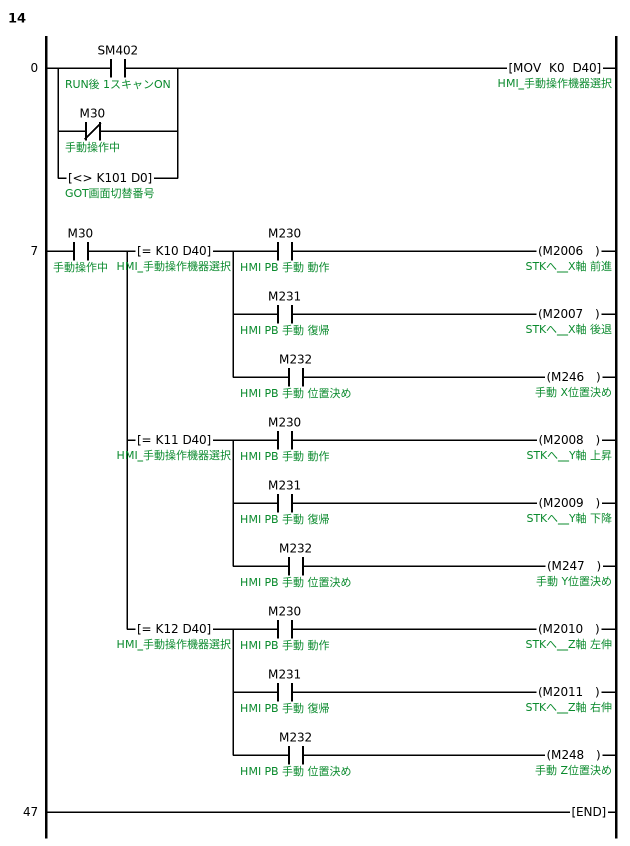
0     LD      SM402  ; RUN後 1スキャンON
      ORI     M30  ; 手動操作中
      OR<>    K101 D0  ; GOT画面切替番号
      MOV     K0 D40  ; HMI_手動操作機器選択
7     LD      M30  ; 手動操作中
      MPS
      AND=    K10 D40  ; HMI_手動操作機器選択
      MPS
      AND     M230  ; HMI PB 手動 動作
      OUT     M2006  ; STKへ__X軸 前進
      MRD
      AND     M231  ; HMI PB 手動 復帰
      OUT     M2007  ; STKへ__X軸 後退
      MPP
      AND     M232  ; HMI PB 手動 位置決め
      OUT     M246  ; 手動 X位置決め
      MRD
      AND=    K11 D40  ; HMI_手動操作機器選択
      MPS
      AND     M230  ; HMI PB 手動 動作
      OUT     M2008  ; STKへ__Y軸 上昇
      MRD
      AND     M231  ; HMI PB 手動 復帰
      OUT     M2009  ; STKへ__Y軸 下降
      MPP
      AND     M232  ; HMI PB 手動 位置決め
      OUT     M247  ; 手動 Y位置決め
      MPP
      AND=    K12 D40  ; HMI_手動操作機器選択
      MPS
      AND     M230  ; HMI PB 手動 動作
      OUT     M2010  ; STKへ__Z軸 左伸
      MRD
      AND     M231  ; HMI PB 手動 復帰
      OUT     M2011  ; STKへ__Z軸 右伸
      MPP
      AND     M232  ; HMI PB 手動 位置決め
      OUT     M248  ; 手動 Z位置決め
47    END
END_PROGRAM

PROGRAM 15  // CV
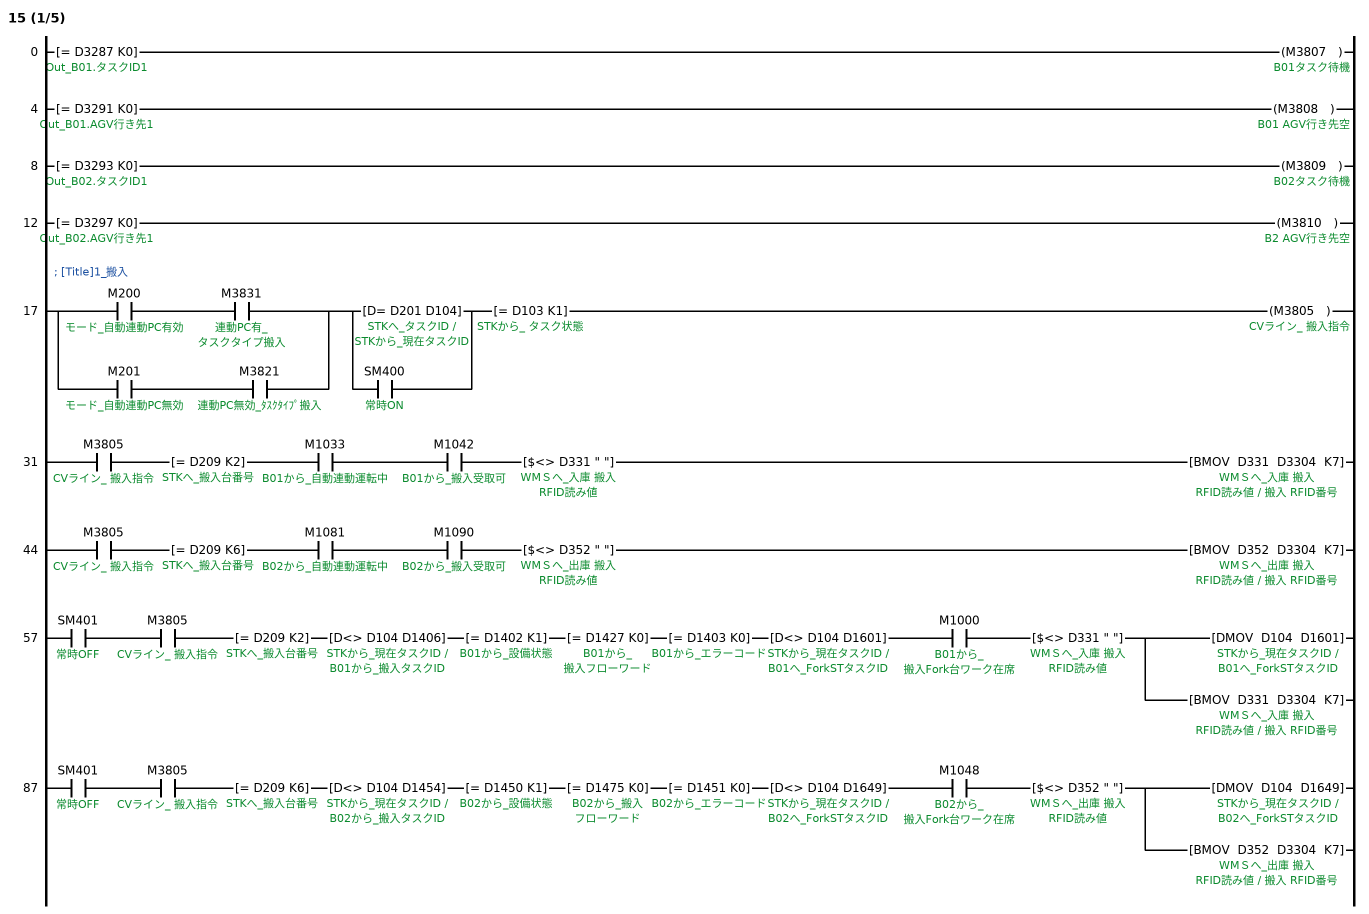
0     LD=     D3287 K0  ; Out_B01.タスクID1
      OUT     M3807  ; B01タスク待機
4     LD=     D3291 K0  ; Out_B01.AGV行き先1
      OUT     M3808  ; B01 AGV行き先空
8     LD=     D3293 K0  ; Out_B02.タスクID1
      OUT     M3809  ; B02タスク待機
12    LD=     D3297 K0  ; Out_B02.AGV行き先1
      OUT     M3810  ; B2 AGV行き先空
; [Title]1_搬入
17    LD      M200  ; モード_自動連動PC有効
      AND     M3831  ; 連動PC有_タスクタイプ搬入
      LD      M201  ; モード_自動連動PC無効
      AND     M3821  ; 連動PC無効_ﾀｽｸﾀｲﾌﾟ搬入
      ORB
      LDD=    D201 D104  ; STKへ_タスクID / STKから_現在タスクID
      OR      SM400  ; 常時ON
      ANB
      AND=    D103 K1  ; STKから_ タスク状態
      OUT     M3805  ; CVライン_ 搬入指令
31    LD      M3805  ; CVライン_ 搬入指令
      AND=    D209 K2  ; STKへ_搬入台番号
      AND     M1033  ; B01から_自動連動運転中
      AND     M1042  ; B01から_搬入受取可
      AND$<>  D331 ""  ; WMＳへ_入庫 搬入 RFID読み値
      BMOV    D331 D3304 K7  ; 搬入 RFID番号
44    LD      M3805  ; CVライン_ 搬入指令
      AND=    D209 K6  ; STKへ_搬入台番号
      AND     M1081  ; B02から_自動連動運転中
      AND     M1090  ; B02から_搬入受取可
      AND$<>  D352 ""  ; WMＳへ_出庫 搬入 RFID読み値
      BMOV    D352 D3304 K7
57    LD      SM401  ; 常時OFF
      AND     M3805  ; CVライン_ 搬入指令
      AND=    D209 K2  ; STKへ_搬入台番号
      ANDD<>  D104 D1406  ; STKから_現在タスクID / B01から_搬入タスクID
      AND=    D1402 K1  ; B01から_設備状態
      AND=    D1427 K0  ; B01から_搬入フローワード
      AND=    D1403 K0  ; B01から_エラーコード
      ANDD<>  D104 D1601  ; STKから_現在タスクID / B01へ_ForkSTタスクID
      AND     M1000  ; B01から_搬入Fork台ワーク在席
      AND$<>  D331 ""  ; WMＳへ_入庫 搬入 RFID読み値
      DMOV    D104 D1601
      BMOV    D331 D3304 K7
87    LD      SM401  ; 常時OFF
      AND     M3805  ; CVライン_ 搬入指令
      AND=    D209 K6  ; STKへ_搬入台番号
      ANDD<>  D104 D1454  ; STKから_現在タスクID / B02から_搬入タスクID
      AND=    D1450 K1  ; B02から_設備状態
      AND=    D1475 K0  ; B02から_搬入 フローワード
      AND=    D1451 K0  ; B02から_エラーコード
      ANDD<>  D104 D1649  ; STKから_現在タスクID / B02へ_ForkSTタスクID
      AND     M1048  ; B02から_搬入Fork台ワーク在席
      AND$<>  D352 ""  ; WMＳへ_出庫 搬入 RFID読み値
      DMOV    D104 D1649
      BMOV    D352 D3304 K7
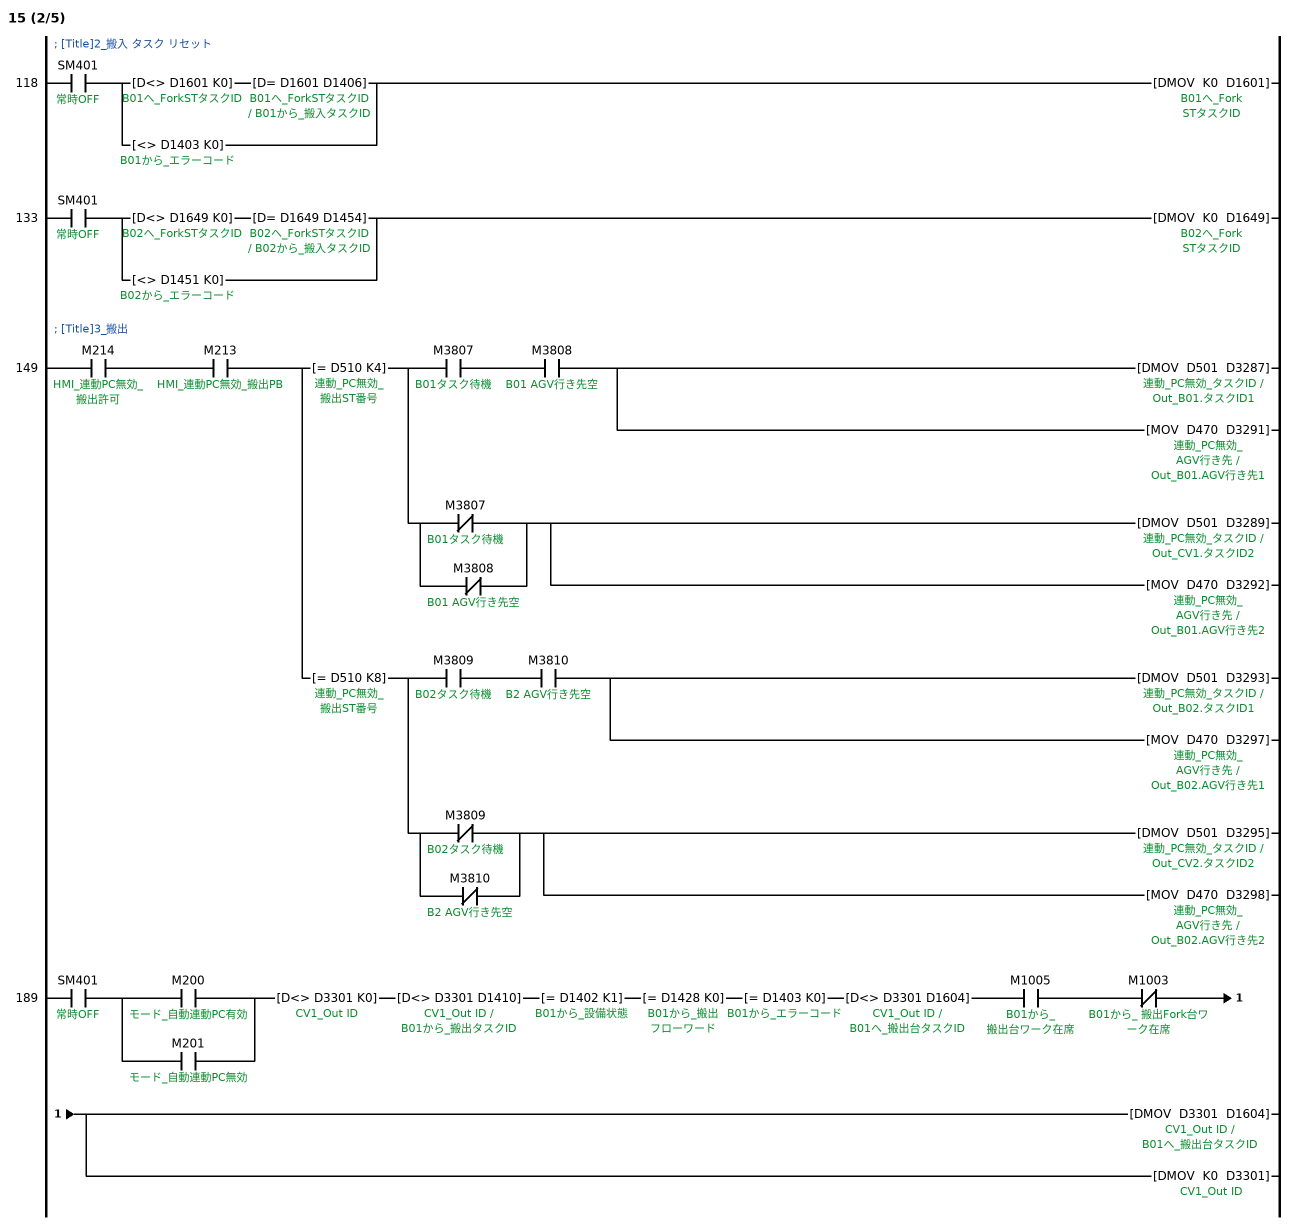
; [Title]2_搬入 タスク リセット
118   LD      SM401  ; 常時OFF
      LDD<>   D1601 K0  ; B01へ_ForkSTタスクID
      ANDD=   D1601 D1406  ; B01へ_ForkSTタスクID / B01から_搬入タスクID
      OR<>    D1403 K0  ; B01から_エラーコード
      ANB
      DMOV    K0 D1601
133   LD      SM401  ; 常時OFF
      LDD<>   D1649 K0  ; B02へ_ForkSTタスクID
      ANDD=   D1649 D1454  ; B02へ_ForkSTタスクID / B02から_搬入タスクID
      OR<>    D1451 K0  ; B02から_エラーコード
      ANB
      DMOV    K0 D1649
; [Title]3_搬出
149   LD      M214  ; HMI_連動PC無効_搬出許可
      AND     M213  ; HMI_連動PC無効_搬出PB
      MPS
      AND=    D510 K4  ; 連動_PC無効_搬出ST番号
      MPS
      AND     M3807  ; B01タスク待機
      AND     M3808  ; B01 AGV行き先空
      DMOV    D501 D3287  ; 連動_PC無効_タスクID
      MOV     D470 D3291  ; 連動_PC無効_AGV行き先
      MPP
      LDI     M3807  ; B01タスク待機
      ORI     M3808  ; B01 AGV行き先空
      ANB
      DMOV    D501 D3289  ; Out_CV1.タスクID2
      MOV     D470 D3292  ; Out_B01.AGV行き先2
      MPP
      AND=    D510 K8  ; 連動_PC無効_搬出ST番号
      MPS
      AND     M3809  ; B02タスク待機
      AND     M3810  ; B2 AGV行き先空
      DMOV    D501 D3293
      MOV     D470 D3297
      MPP
      LDI     M3809  ; B02タスク待機
      ORI     M3810  ; B2 AGV行き先空
      ANB
      DMOV    D501 D3295  ; Out_CV2.タスクID2
      MOV     D470 D3298  ; Out_B02.AGV行き先2
189   LD      SM401  ; 常時OFF
      LD      M200  ; モード_自動連動PC有効
      OR      M201  ; モード_自動連動PC無効
      ANB
      ANDD<>  D3301 K0  ; CV1_Out ID
      ANDD<>  D3301 D1410  ; CV1_Out ID / B01から_搬出タスクID
      AND=    D1402 K1  ; B01から_設備状態
      AND=    D1428 K0  ; B01から_搬出 フローワード
      AND=    D1403 K0  ; B01から_エラーコード
      ANDD<>  D3301 D1604  ; CV1_Out ID / B01へ_搬出台タスクID
      AND     M1005  ; B01から_ 搬出台ワーク在席
      ANI     M1003  ; B01から_ 搬出Fork台ワーク在席
      DMOV    D3301 D1604
      DMOV    K0 D3301
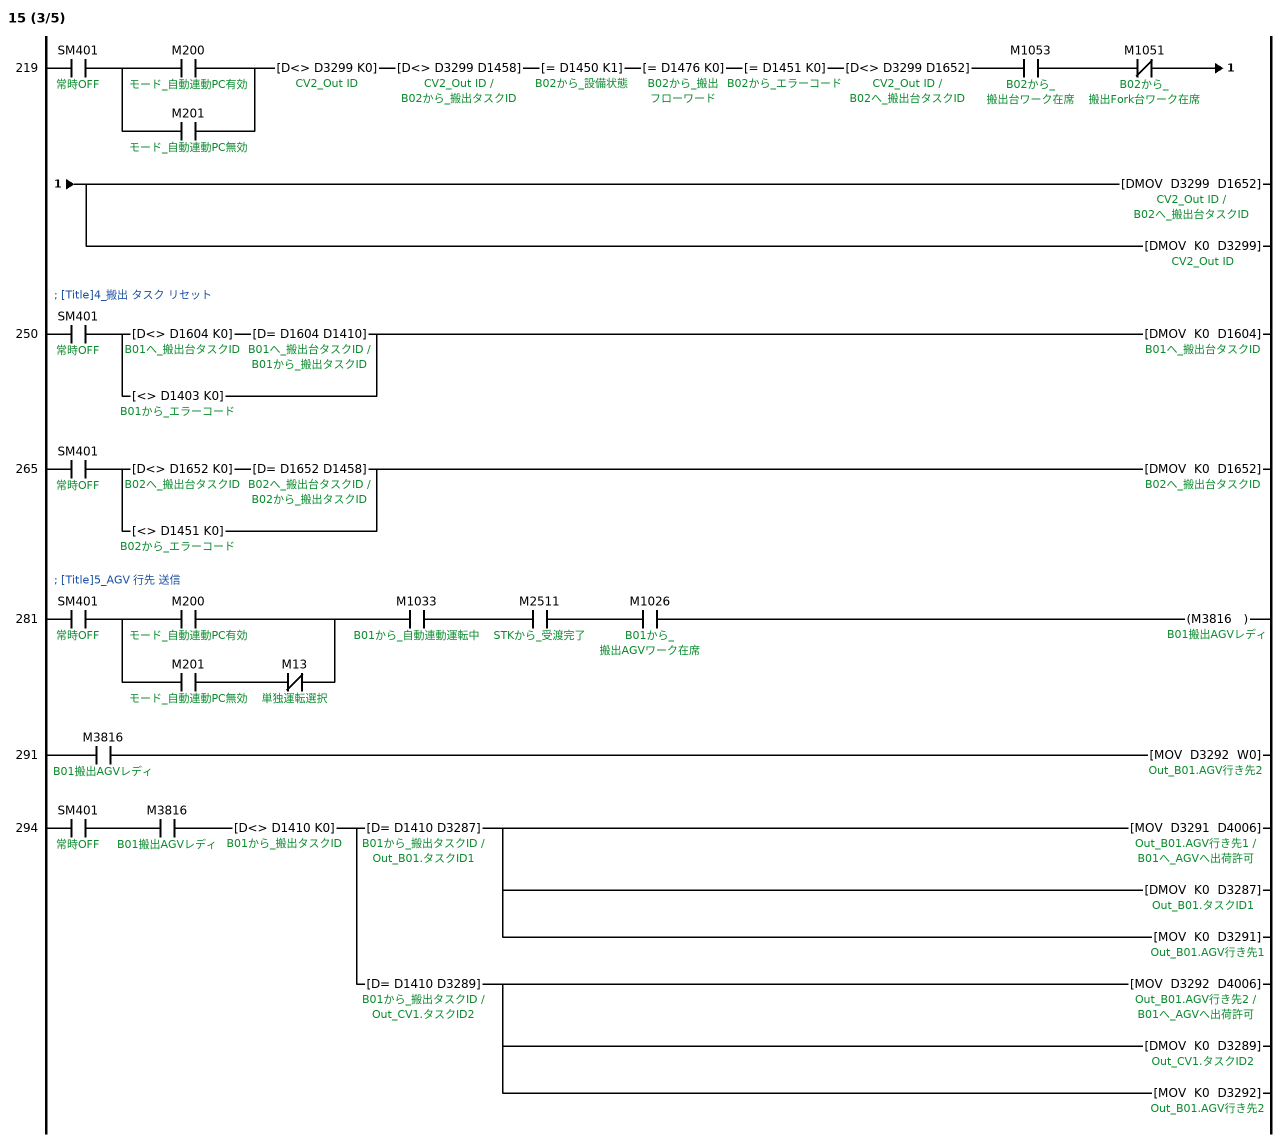
219   LD      SM401  ; 常時OFF
      LD      M200  ; モード_自動連動PC有効
      OR      M201  ; モード_自動連動PC無効
      ANB
      ANDD<>  D3299 K0  ; CV2_Out ID
      ANDD<>  D3299 D1458  ; CV2_Out ID / B02から_搬出タスクID
      AND=    D1450 K1  ; B02から_設備状態
      AND=    D1476 K0  ; B02から_搬出 フローワード
      AND=    D1451 K0  ; B02から_エラーコード
      ANDD<>  D3299 D1652  ; CV2_Out ID / B02へ_搬出台タスクID
      AND     M1053  ; B02から_搬出台ワーク在席
      ANI     M1051  ; B02から_搬出Fork台ワーク在席
      DMOV    D3299 D1652
      DMOV    K0 D3299
; [Title]4_搬出 タスク リセット
250   LD      SM401  ; 常時OFF
      LDD<>   D1604 K0  ; B01へ_搬出台タスクID
      ANDD=   D1604 D1410  ; B01へ_搬出台タスクID / B01から_搬出タスクID
      OR<>    D1403 K0  ; B01から_エラーコード
      ANB
      DMOV    K0 D1604
265   LD      SM401  ; 常時OFF
      LDD<>   D1652 K0  ; B02へ_搬出台タスクID
      ANDD=   D1652 D1458  ; B02へ_搬出台タスクID / B02から_搬出タスクID
      OR<>    D1451 K0  ; B02から_エラーコード
      ANB
      DMOV    K0 D1652
; [Title]5_AGV 行先 送信
281   LD      SM401  ; 常時OFF
      LD      M200  ; モード_自動連動PC有効
      LD      M201  ; モード_自動連動PC無効
      ANI     M13  ; 単独運転選択
      ORB
      ANB
      AND     M1033  ; B01から_自動連動運転中
      AND     M2511  ; STKから_受渡完了
      AND     M1026  ; B01から_搬出AGVワーク在席
      OUT     M3816  ; B01搬出AGVレディ
291   LD      M3816  ; B01搬出AGVレディ
      MOV     D3292 W0
294   LD      SM401  ; 常時OFF
      AND     M3816  ; B01搬出AGVレディ
      ANDD<>  D1410 K0  ; B01から_搬出タスクID
      MPS
      ANDD=   D1410 D3287  ; B01から_搬出タスクID / Out_B01.タスクID1
      MOV     D3291 D4006  ; B01へ_AGVへ出荷許可
      DMOV    K0 D3287
      MOV     K0 D3291
      MPP
      ANDD=   D1410 D3289  ; B01から_搬出タスクID / Out_CV1.タスクID2
      MOV     D3292 D4006
      DMOV    K0 D3289
      MOV     K0 D3292
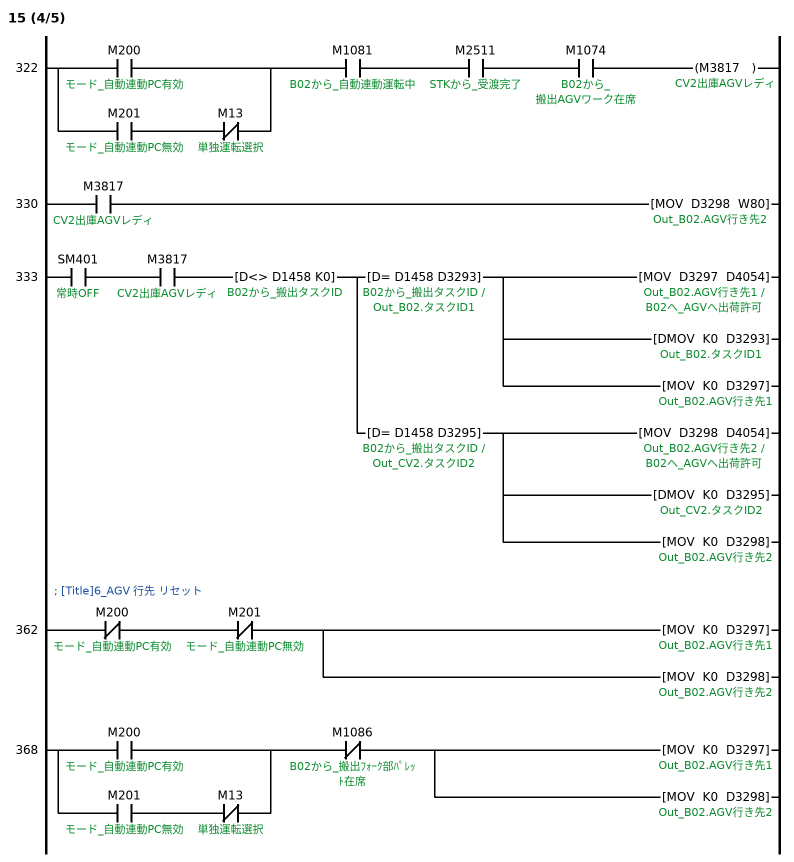
322   LD      M200  ; モード_自動連動PC有効
      LD      M201  ; モード_自動連動PC無効
      ANI     M13  ; 単独運転選択
      ORB
      AND     M1081  ; B02から_自動連動運転中
      AND     M2511  ; STKから_受渡完了
      AND     M1074  ; B02から_搬出AGVワーク在席
      OUT     M3817  ; CV2出庫AGVレディ
330   LD      M3817  ; CV2出庫AGVレディ
      MOV     D3298 W80
333   LD      SM401  ; 常時OFF
      AND     M3817  ; CV2出庫AGVレディ
      ANDD<>  D1458 K0  ; B02から_搬出タスクID
      MPS
      ANDD=   D1458 D3293  ; B02から_搬出タスクID / Out_B02.タスクID1
      MOV     D3297 D4054  ; B02へ_AGVへ出荷許可
      DMOV    K0 D3293
      MOV     K0 D3297
      MPP
      ANDD=   D1458 D3295  ; B02から_搬出タスクID / Out_CV2.タスクID2
      MOV     D3298 D4054
      DMOV    K0 D3295
      MOV     K0 D3298
; [Title]6_AGV 行先 リセット
362   LDI     M200  ; モード_自動連動PC有効
      ANI     M201  ; モード_自動連動PC無効
      MOV     K0 D3297
      MOV     K0 D3298
368   LD      M200  ; モード_自動連動PC有効
      LD      M201  ; モード_自動連動PC無効
      ANI     M13  ; 単独運転選択
      ORB
      ANI     M1086  ; B02から_搬出ﾌｫｰｸ部ﾊﾟﾚｯﾄ在席
      MOV     K0 D3297
      MOV     K0 D3298
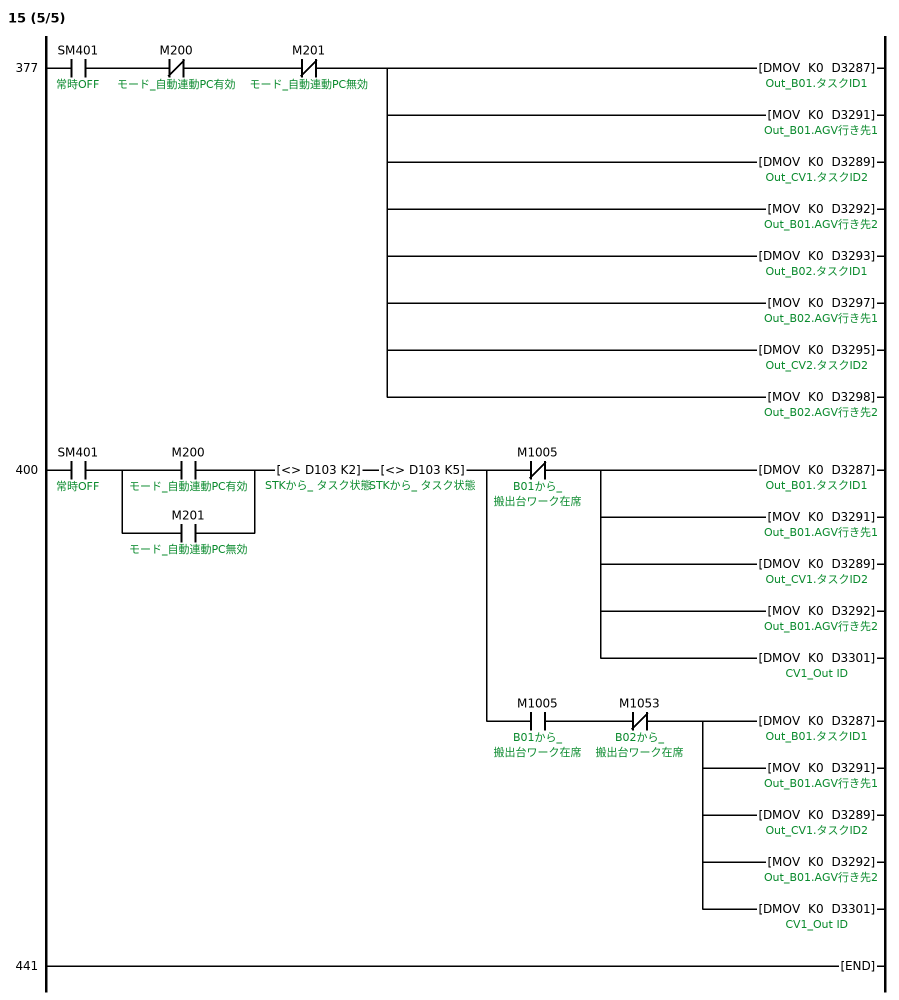
377   LD      SM401  ; 常時OFF
      ANI     M200  ; モード_自動連動PC有効
      ANI     M201  ; モード_自動連動PC無効
      DMOV    K0 D3287
      MOV     K0 D3291
      DMOV    K0 D3289
      MOV     K0 D3292
      DMOV    K0 D3293
      MOV     K0 D3297
      DMOV    K0 D3295
      MOV     K0 D3298
400   LD      SM401  ; 常時OFF
      LD      M200  ; モード_自動連動PC有効
      OR      M201  ; モード_自動連動PC無効
      ANB
      AND<>   D103 K2  ; STKから_ タスク状態
      AND<>   D103 K5  ; STKから_ タスク状態
      MPS
      ANI     M1005  ; B01から_ 搬出台ワーク在席
      DMOV    K0 D3287
      MOV     K0 D3291
      DMOV    K0 D3289
      MOV     K0 D3292
      DMOV    K0 D3301
      MPP
      AND     M1005  ; B01から_ 搬出台ワーク在席
      ANI     M1053  ; B02から_搬出台ワーク在席
      DMOV    K0 D3287
      MOV     K0 D3291
      DMOV    K0 D3289
      MOV     K0 D3292
      DMOV    K0 D3301
441   END
END_PROGRAM

PROGRAM 20  // 在庫データ管理
VAR
  AO1 : INT;
  AO2 : INT;
  AO3 : DINT;
  Temp : BOOL;
  RFIE_Len : INT;
  QA : INT;
END_VAR
(*1_在庫更新*)
(*2_空き保管場所検索*)
(*3_在庫クリア*)
(*4_库存查询*)	
(*5_搬出後在庫整理*)
(*6_搬入完了*)
(*7_移庫*)

(*----------------------------------------------ソフト要素入力自動割り当て----------------------------------------------*)
DMOV(TRUE,D3301,B01CV_OutID);
DMOV(TRUE,D3229,B02CV_OutID);
BMOV(TRUE,D3304,K7,搬入RFID_Coding);
(*-------------------------------------------------------------------------------------------------------------------*)

(*1_在庫更新*)
 AO1:=0;
 AO2:=0;
FOR AO1:=1 TO 14 DO
	FOR AO2:=1 TO 5 DO
	    IF  inventory_1[ AO1].層[AO2]<>'' AND inventory_1[ AO1].層[AO2]<>'            ' THEN
			inventory_Bit1[AO1].層[AO2]:=TRUE;
		ELSE
			inventory_Bit1[AO1].層[AO2]:=FALSE;
		END_IF;
		
		IF  inventory_2[ AO1].層[AO2]<>'' AND inventory_2[ AO1].層[AO2]<>'            '  THEN
			inventory_Bit2[AO1].層[AO2]:=TRUE;
		ELSE
			inventory_Bit2[AO1].層[AO2]:=FALSE;
		END_IF;
	END_FOR;
END_FOR;

(*2_空き保管場所検索*)
Temp:=FALSE;
IF Single_Machine.空き保管場所検索 AND Mode=1 THEN
	 AO1:=0;
     AO2:=0;
     Alone.Task_Type:=1;
    FOR AO1:=1 TO 14 DO
	    FOR AO2:=1 TO 5 DO
	     	IF inventory_Bit1[AO1].層[AO2]=FALSE THEN
			     Alone.終点棚:=1;
			     Alone.終点列:=AO1;
			     Alone.終点層:=AO2;
			     Temp:=TRUE;
			    EXIT;
	     	END_IF;
	     	IF inventory_Bit2[AO1].層[AO2]=FALSE THEN
			     Alone.終点棚:=2;
			     Alone.終点列:=AO1;
			     Alone.終点層:=AO2;
			     Temp:=TRUE;
			    EXIT;
	     	END_IF;
	    END_FOR;
	    IF Temp THEN
	    	EXIT;
	    END_IF;
	END_FOR;	
END_IF;

(*3_在庫クリア*)
IF 在庫クリア THEN
	 AO1:=0;
     AO2:=0;
	FOR AO1:=1 TO 14 DO
		FOR AO2:=1 TO 5 DO
			  inventory_1[ AO1].層[AO2]:='';
			  inventory_2[ AO1].層[AO2]:='';
		END_FOR;
	END_FOR;
END_IF;

(*4_在庫確認*)	
IF Single_Machine.Query AND Single_Machine.成功=FALSE AND Single_Machine.失敗=FALSE THEN
	Single_Machine.棚場所:=0;
	Single_Machine.列場所:=0;
	Single_Machine.層場所:=0;
	Alone.Task_Type:=2;
	AO1:=0;
    AO2:=0;
	FOR AO1:=1 TO 14 DO
		FOR AO2:=1 TO 5 DO
			IF Single_Machine.RFID入力= inventory_1[ AO1].層[AO2] THEN
				Single_Machine.棚場所:=1;
				Single_Machine.列場所:=AO1;
				Single_Machine.層場所:=AO2;
				Single_Machine.成功:=TRUE;
				Single_Machine.失敗:=FALSE;
				Alone.起点棚:=Single_Machine.棚場所;
                Alone.起点列:=Single_Machine.列場所;
                Alone.起点層:=Single_Machine.層場所;
				EXIT;
			END_IF;
			IF Single_Machine.RFID入力= inventory_2[ AO1].層[AO2] THEN
				Single_Machine.棚場所:=2;
				Single_Machine.列場所:=AO1;
				Single_Machine.層場所:=AO2;
				Single_Machine.成功:=TRUE;
				Single_Machine.失敗:=FALSE;
				Alone.起点棚:=Single_Machine.棚場所;
                Alone.起点列:=Single_Machine.列場所;
                Alone.起点層:=Single_Machine.層場所;
				EXIT;
			END_IF;
			
			IF AO1=14 AND AO2=5 THEN
	         	Single_Machine.失敗:=TRUE;
		        Single_Machine.成功:=FALSE;
		        Single_Machine.棚場所:=0;
				Single_Machine.列場所:=0;
				Single_Machine.層場所:=0;
				Alone.起点棚:=Single_Machine.棚場所;
                Alone.起点列:=Single_Machine.列場所;
                Alone.起点層:=Single_Machine.層場所;
			END_IF;
		END_FOR;
		IF Single_Machine.成功 THEN
			EXIT;
		END_IF;
	END_FOR;
END_IF;

OUT_T(Single_Machine.Query=FALSE AND (Single_Machine.成功 OR Single_Machine.失敗),TC2,30);
IF   TC2 THEN
	   (*rst(TS2,TC2);*)
	  Single_Machine.失敗:=FALSE;
	  Single_Machine.成功:=FALSE;
END_IF;	

IF  Stacker_R.Task_Status=5 AND NOT Stacker_Done THEN
	
(*5_搬出後在庫整理*)
  IF Stacker_W.Task_Type=2 AND Stacker_W.Task_ID=Stacker_R.現在Task_ID AND Stacker_R.Task_Status=5 THEN
   	IF Stacker_W.起点棚=1 THEN
   		 inventory_1[ Stacker_W.起点列].層[Stacker_W.起点層]:= '';
   	ELSIF
   		Stacker_W.起点棚=2 THEN
   		inventory_2[ Stacker_W.起点列].層[Stacker_W.起点層]:= '';
   	END_IF;
   	
   	IF Stacker_W.搬出ST_NO=3 AND B01CV_OutID<>Stacker_R.現在Task_ID THEN
   		B01CV_OutID:=Stacker_R.現在Task_ID;
   	ELSIF
   		Stacker_W.搬出ST_NO=4 AND B02CV_OutID<>Stacker_R.現在Task_ID THEN
   		B02CV_OutID:=Stacker_R.現在Task_ID;   	
   		END_IF;
  END_IF;
    	
(*6_搬入完了*)
   IF   Stacker_W.Task_Type=1 AND Stacker_W.Task_ID=Stacker_R.現在Task_ID AND Stacker_R.Task_Status=5 AND 搬入RFID_Coding<> '' THEN     
          IF Stacker_W.終点棚=1 THEN
          	 inventory_1[ Stacker_W.終点列].層[Stacker_W.終点層]:=搬入RFID_Coding;
          	 搬入RFID_Coding:= '' ;
          ELSIF 
          	Stacker_W.終点棚=2  THEN
          	 inventory_2[ Stacker_W.終点列].層[Stacker_W.終点層]:=搬入RFID_Coding;
          	 搬入RFID_Coding:= '' ;
          END_IF;
  END_IF;
 
 (*7_移庫*)
  IF  Stacker_W.Task_Type=3 AND Stacker_W.Task_ID=Stacker_R.現在Task_ID AND Stacker_R.Task_Status=5 THEN   
          IF Stacker_W.終点棚=1 THEN
          	  IF Stacker_W.起点棚=1 THEN
          	      inventory_1[ Stacker_W.終点列].層[Stacker_W.終点層]:=inventory_1[ Stacker_W.起点列].層[Stacker_W.起点層];
          	      inventory_1[ Stacker_W.起点列].層[Stacker_W.起点層]:= '';
          	  ELSIF Stacker_W.起点棚=2 THEN
   		          inventory_1[ Stacker_W.終点列].層[Stacker_W.終点層]:=inventory_2[ Stacker_W.起点列].層[Stacker_W.起点層];
   		           inventory_2[ Stacker_W.起点列].層[Stacker_W.起点層]:= '';
          	  END_IF;
          	  
          ELSIF Stacker_W.終点棚=2 THEN
          	 IF Stacker_W.起点棚=1 THEN
          	      inventory_2[ Stacker_W.終点列].層[Stacker_W.終点層]:=inventory_1[ Stacker_W.起点列].層[Stacker_W.起点層];
          	      inventory_1[ Stacker_W.起点列].層[Stacker_W.起点層]:= '';
          	  ELSIF Stacker_W.起点棚=2 THEN
   		          inventory_2[ Stacker_W.終点列].層[Stacker_W.終点層]:=inventory_2[ Stacker_W.起点列].層[Stacker_W.起点層];
   		           inventory_2[ Stacker_W.起点列].層[Stacker_W.起点層]:= '';
          	  END_IF;
          END_IF;
   END_IF;
END_IF; 	
Stacker_Done:= Stacker_R.Task_Status=5 ;

(*----------------------------------------------ソフト要素出力自動的割り当て----------------------------------------------*)
DMOV(TRUE,B01CV_OutID,D3301);
DMOV(TRUE,B02CV_OutID,D3229);
BMOV(TRUE,搬入RFID_Coding,K7,D3304);
(*---------------------------------------------------------------------------------------------------------------------*)
END_PROGRAM

PROGRAM 40  // PLC 出力
